// TIA Portal project "Mmot_20230531_1041" (V15.1)

(* hardware
DEVICE "S7-1200 station_1"  S7-1200 Station
   slot 0: "Rack_0"  S7-1200 Rack  Rack  V1.0
   slot 1: "PLC_1"  CPU 1214C DC/DC/DC  6ES7 214-1AG40-0XB0  V4.3
   slot 2: "DI 8x24VDC_1"  6ES7 221-1BF32-0XB0  V2.0
*)

// ===== PLC "PLC_1"  CPU 1214C DC/DC/DC =====

VAR_GLOBAL   // PLC tag table "Default tag table"
   "System_Byte" AT %MB1 : Byte;
   "FirstScan" AT %M1.0 : Bool;
   "DiagStatusUpdate" AT %M1.1 : Bool;
   "AlwaysTRUE" AT %M1.2 : Bool;
   "AlwaysFALSE" AT %M1.3 : Bool;
   "Clock_Byte" AT %MB0 : Byte;
   "Clock_10Hz" AT %M0.0 : Bool;
   "Clock_5Hz" AT %M0.1 : Bool;
   "Clock_2.5Hz" AT %M0.2 : Bool;
   "Clock_2Hz" AT %M0.3 : Bool;
   "Clock_1.25Hz" AT %M0.4 : Bool;
   "Clock_1Hz" AT %M0.5 : Bool;
   "Clock_0.625Hz" AT %M0.6 : Bool;
   "Clock_0.5Hz" AT %M0.7 : Bool;
   "Detector_Axis_Step" AT %Q0.3 : Bool;
   "Doors_Axis_Pulse" AT %Q0.0 : Bool;
   "start" AT %M3.0 : Bool;
   "button_forward" AT %I1.2 : Bool;
   "button_back" AT %I1.3 : Bool;
   "Detector_Axis_Direction" AT %Q0.5 : Bool;
   "Source_Axis_Pulse" AT %Q0.2 : Bool;
   "Source_Axis_Direction" AT %Q0.4 : Bool;
   "Doors_Axis_Direction" AT %Q0.6 : Bool;
   "Roll_Axis_Pulse" AT %Q0.1 : Bool;
   "Roll_Axis_Direction" AT %Q0.7 : Bool;
   "MEMO-1" AT %M10.1 : Bool;
   "MEMO-2" AT %M10.2 : Bool;
END_VAR

VAR_GLOBAL   // PLC tag table "SwitchLimits"
   "SL3A" AT %I0.5 : Bool;
   "SL3B" AT %I0.6 : Bool;
   "SL1A" AT %I0.0 : Bool;
   "SL1B" AT %I0.1 : Bool;
   "SL1C" AT %I0.2 : Bool;
   "SL2A" AT %I0.3 : Bool;
   "SL2B" AT %I0.4 : Bool;
   "SL4A" AT %I0.7 : Bool;
   "SL5" AT %I8.4 : Bool;
   "SL6" AT %I8.5 : Bool;
END_VAR

VAR_GLOBAL   // PLC tag table "source_control"
   "source_block" AT %Q1.0 : Bool;
   "radiation_lamp" AT %Q1.1 : Bool;
   "power_enabled" AT %I1.4 : Bool;
   "emitting" AT %I1.5 : Bool;
END_VAR

VAR_GLOBAL   // PLC tag table "general"
   "S1_alarm" AT %I8.0 : Bool;
   "S2_alarm" AT %I8.1 : Bool;
   "S3_alarm" AT %I8.2 : Bool;
   "S4_alarm" AT %I8.3 : Bool;
   "Q1_control" AT %I1.0 : Bool;
   "Q2_control" AT %I1.1 : Bool;
   "E_button_pressed" AT %M10.0 : Bool;
   "moveC" AT %MW10 : Int;
END_VAR

TYPE "TCON_IP_v42"
   STRUCT
      InterfaceID : Hw_Any;
      ID : Conn_Ouc;
      ConnectionType : Byte := 11;
      ActiveEstablished : Bool := FALSE;
      RemoteAddress : Array[1..4] of Byte;
      RemotePort : UInt := 0;
      LocalPort : UInt := 502;
   END_STRUCT;
   // RemoteAddress[1] := 0;
   // RemoteAddress[2] := 0;
   // RemoteAddress[3] := 0;
   // RemoteAddress[4] := 0;
END_TYPE

DATA_BLOCK "MB_Regs"   // DB2
{ S7_Optimized_Access := 'FALSE' }
VERSION : 0.1
   VAR
      data : Array[0..79] of Word;
   END_VAR
BEGIN
   data[0] := 1;   // 1 Вкл, 0 Выкл
   data[1] := 0;   // 1 - калибровка
   data[2] := 0;   // вращение туда
   data[3] := 0;   // вращение сюда
   data[4] := 0;   // Позиция ст слово
   // data[5] : Позиция мл Слово
   // data[6] : Скорость
   // data[8] : Тек поз ст
   // data[9] : Тек поз мл
   // data[10] : Статус
   // data[11] : Ошибка
   // data[12] : Калибровано
   // data[7] : Сброс
   // data[13] : Halt
   // data[14] : move_to_abs_pos
   // data[15] : move_to_rel_pos
   // data[20] : 1 Вкл, 0 Выкл
   // data[21] : 1 - калибровка
   // data[22] : вращение туда
   // data[23] : вращение сюда
   // data[24] : Позиция ст слово
   // data[25] : Позиция мл Слово
   // data[26] : Скорость
   // data[27] : Сброс
   // data[28] : Тек поз ст
   // data[29] : Тек поз мл
   // data[30] : Статус
   // data[31] : Ошибка
   // data[32] : Калибровано
   // data[33] : Halt
   // data[34] : move_to_abs_pos
   // data[35] : move_to_rel_pos
   // data[40] : 1 Вкл, 0 Выкл
   // data[41] : 1 - калибровка
   // data[42] : вращение туда
   // data[43] : вращение сюда
   // data[44] : Позиция ст слово
   // data[45] : Позиция мл Слово
   // data[46] : Скорость
   // data[47] : Сброс
   // data[48] : Тек поз ст
   // data[49] : Тек поз мл
   // data[50] : Статус
   // data[51] : Ошибка
   // data[52] : Калибровано
   // data[53] : Halt
   // data[54] : move_to_abs_pos
   // data[55] : move_to_rel_pos
   // data[60] : 1 Вкл, 0 Выкл
   // data[61] : 1 - калибровка
   // data[62] : вращение туда
   // data[63] : вращение сюда
   // data[64] : Позиция ст слово
   // data[65] : Позиция мл Слово
   // data[66] : Скорость
   // data[67] : Сброс
   // data[68] : Тек поз ст
   // data[69] : Тек поз мл
   // data[70] : Статус
   // data[71] : Ошибка
   // data[72] : Калибровано
   // data[73] : Halt
   // data[74] : move_to_abs_pos
   // data[75] : move_to_rel_pos
   // data[19] : Block_is_active
   // data[16] : Emission_active
   // data[17] : Power_enabled
   // data[18] : E_stop_button_pressed
   // data[36] : limit1
   // data[37] : limit2
   // data[56] : limit1
   // data[57] : limit2
   // data[76] : moveFrame
   // data[77] : moveCounter
END_DATA_BLOCK

DATA_BLOCK "connect"   // DB3
{ S7_Optimized_Access := 'TRUE' }
VERSION : 0.1
   VAR
      con : "TCON_IP_v42";
      connect : TCON_IP_v4;
   END_VAR
BEGIN
   con.InterfaceID := 64;
   con.ID := 1;
   connect.InterfaceId := 64;
   connect.ID := 1;
   connect.ConnectionType := 11;
   connect.LocalPort := 502;
END_DATA_BLOCK

DATA_BLOCK "door_axe_DB"   // DB6
{ S7_Optimized_Access := 'TRUE' }
VERSION : 0.1
// stored: InstanceOfName door_axe
"door_axe"
BEGIN
END_DATA_BLOCK

DATA_BLOCK "TCP_motion_control_DB"   // DB14
{ S7_Optimized_Access := 'TRUE' }
VERSION : 0.1
// stored: InstanceOfName TCP_motion_control
"TCP_motion_control"
BEGIN
END_DATA_BLOCK

DATA_BLOCK "detector_axe_DB"   // DB15
{ S7_Optimized_Access := 'TRUE' }
VERSION : 0.1
// stored: InstanceOfName detector_axe
"detector_axe"
BEGIN
END_DATA_BLOCK

DATA_BLOCK "source_axe_DB"   // DB17
{ S7_Optimized_Access := 'TRUE' }
VERSION : 0.1
// stored: InstanceOfName source_axe
"source_axe"
BEGIN
END_DATA_BLOCK

DATA_BLOCK "roll_axe_DB"   // DB38
{ S7_Optimized_Access := 'TRUE' }
VERSION : 0.1
// stored: InstanceOfName roll_axe
"roll_axe"
BEGIN
END_DATA_BLOCK

DATA_BLOCK "safety_DB"   // DB40
{ S7_Optimized_Access := 'TRUE' }
VERSION : 0.1
// stored: InstanceOfName safety
"safety"
BEGIN
END_DATA_BLOCK

DATA_BLOCK "CalibrationData"   // DB41
{ S7_Optimized_Access := 'FALSE' }
VERSION : 0.1
   VAR
      Axe1_calibrated : Bool;
      Axe2_calibrated : Bool;
      Axe3_calibrated : Bool;
      Axe4_calibrated : Bool;
      Axe1_saved_pos : Real;
      Axe2_saved_pos : Real;
      Axe3_saved_pos : Real;
      Axe4_saved_pos : Real;
   END_VAR
BEGIN
END_DATA_BLOCK

DATA_BLOCK "safe_done"   // DB47
{ S7_Optimized_Access := 'TRUE' }
VERSION : 0.1
   VAR
      Axe1_SU_calibration_done : Bool;
      Axe2_SU_calibration_done : Bool;
      Axe3_SU_calibration_done : Bool;
      Axe4_SU_calibration_done : Bool;
      control_position : Real;
      control_position_1 : Real;
      control_position_2 : Real;
   END_VAR
BEGIN
END_DATA_BLOCK

// folder: System blocks/Program resources

DATA_BLOCK "IEC_Timer_0_DB"   // DB46
{ S7_Optimized_Access := 'TRUE' }
AUTHOR : Simatic
FAMILY : IEC
NAME : IEC_TMR
VERSION : 1.0
// stored: InstanceOfName IEC_TIMER
"IEC_TIMER"
BEGIN
END_DATA_BLOCK

DATA_BLOCK "IEC_Timer_0_DB_2"   // DB48
{ S7_Optimized_Access := 'TRUE' }
AUTHOR : Simatic
FAMILY : IEC
NAME : IEC_TMR
VERSION : 1.0
// stored: InstanceOfName IEC_TIMER
"IEC_TIMER"
BEGIN
END_DATA_BLOCK

// folder: (top level)

DATA_BLOCK "Detector_Axis"   // DB4, Motion_DB
{ S7_Optimized_Access := 'TRUE' }
AUTHOR : SIMATIC
FAMILY : BasicMC
NAME : TO_PosAx
VERSION : 6.0
// stored: InstanceOfName TO_PositioningAxis
"TO_PositioningAxis"
BEGIN
   // Axis.PassiveHomingReferencePointSwitch_AddressCU = %I0.5
   // Axis.HomingReferencePointSwitch_AddressCU = %I0.5
   // Axis.PositionLimitsMax_AddressCU = %I0.6
   // Axis.PositionLimitsMin_AddressCU = %I0.7
   // Axis.DirectionOutputEnabledCU = TRUE
   // Axis.OnlinePtoIndexCU = 2
   // Axis.LengthUnitNormalized.Distance = 1013
   // Axis.OnlinePtoModeCU = 16#0000_0002
   // Axis.SelectedChannel2EnumCU = %Q0.5
   // Axis.SelectedChannel1EnumCU = %Q0.3
   // Pulse.MinDeltaDeltaFrequencyCU = 0.004
   // Pulse.MaxDeltaDeltaFrequencyCU = 1.0E+10
   // Pulse.MinDeltaFrequencyCU = 0.005
   // Pulse.MaxDeltaFrequencyCU = 9.5E+9
   // Pulse.MinFrequencyCU = 1.0
   // Pulse.MaxFrequencyCU = 100000.0
   // Pulse.OutputSourceCU = 16#0000_0000
   // Axis.SelectPTO = 2
END_DATA_BLOCK

DATA_BLOCK "Source_Axis"   // DB5, Motion_DB
{ S7_Optimized_Access := 'TRUE' }
AUTHOR : SIMATIC
FAMILY : BasicMC
NAME : TO_PosAx
VERSION : 6.0
// stored: InstanceOfName TO_PositioningAxis
"TO_PositioningAxis"
BEGIN
   // Axis.PositionLimitsMax_AddressCU = %I0.4
   // Axis.HomingReferencePointSwitch_AddressCU = %I0.3
   // Axis.PassiveHomingReferencePointSwitch_AddressCU = %I0.3
   // Axis.PositionLimitsMin_AddressCU = %I0.3
   // Axis.DirectionOutputEnabledCU = TRUE
   // Axis.OnlinePtoIndexCU = 1
   // Axis.LengthUnitNormalized.Distance = 1013
   // Axis.OnlinePtoModeCU = 16#0000_0002
   // Axis.SelectedChannel2EnumCU = %Q0.4
   // Axis.SelectedChannel1EnumCU = %Q0.2
   // Pulse.MinDeltaDeltaFrequencyCU = 0.004
   // Pulse.MaxDeltaDeltaFrequencyCU = 1.0E+10
   // Pulse.MinDeltaFrequencyCU = 0.005
   // Pulse.MaxDeltaFrequencyCU = 9.5E+9
   // Pulse.MinFrequencyCU = 1.0
   // Pulse.MaxFrequencyCU = 100000.0
   // Pulse.OutputSourceCU = 16#0000_0000
   // Axis.SelectPTO = 1
END_DATA_BLOCK

DATA_BLOCK "Doors_Axis"   // DB16, Motion_DB
{ S7_Optimized_Access := 'TRUE' }
AUTHOR : SIMATIC
FAMILY : BasicMC
NAME : TO_PosAx
VERSION : 6.0
// stored: InstanceOfName TO_PositioningAxis
"TO_PositioningAxis"
BEGIN
   // Axis.PositionLimitsMin_AddressCU = %I0.1
   // Axis.PassiveHomingReferencePointSwitch_AddressCU = %I0.1
   // Axis.PositionLimitsMax_AddressCU = %I0.0
   // Axis.HomingReferencePointSwitch_AddressCU = %I0.1
   // Axis.DirectionOutputEnabledCU = TRUE
   // Axis.LengthUnitNormalized.Distance = 1013
   // Axis.OnlinePtoModeCU = 16#0000_0002
   // Axis.SelectedChannel2EnumCU = %Q0.6
   // Axis.SelectedChannel1EnumCU = %Q0.0
   // Pulse.MinDeltaDeltaFrequencyCU = 0.004
   // Pulse.MaxDeltaDeltaFrequencyCU = 1.0E+10
   // Pulse.MinDeltaFrequencyCU = 0.005
   // Pulse.MaxDeltaFrequencyCU = 9.5E+9
   // Pulse.MinFrequencyCU = 1.0
   // Pulse.MaxFrequencyCU = 100000.0
   // Pulse.OutputSourceCU = 16#0000_0000
   // Axis.SelectPTO = 0
END_DATA_BLOCK

DATA_BLOCK "Roll_Axis"   // DB39, Motion_DB
{ S7_Optimized_Access := 'TRUE' }
AUTHOR : SIMATIC
FAMILY : BasicMC
NAME : TO_PosAx
VERSION : 6.0
// stored: InstanceOfName TO_PositioningAxis
"TO_PositioningAxis"
BEGIN
   // Axis.LengthUnit.LastDistance = -1
   // Axis.OnlinePtoIndexCU = 3
   // Axis.DirectionOutputEnabledCU = TRUE
   // Axis.OnlinePtoModeCU = 16#0000_0002
   // Axis.SelectedChannel2EnumCU = %Q0.7
   // Axis.SelectedChannel1EnumCU = %Q0.1
   // Pulse.MinDeltaDeltaFrequencyCU = 0.004
   // Pulse.MaxDeltaDeltaFrequencyCU = 1.0E+10
   // Pulse.MinDeltaFrequencyCU = 0.005
   // Pulse.MaxDeltaFrequencyCU = 9.5E+9
   // Pulse.MinFrequencyCU = 1.0
   // Pulse.MaxFrequencyCU = 100000.0
   // Pulse.OutputSourceCU = 16#0000_0000
   // Axis.SelectPTO = 3
END_DATA_BLOCK

FUNCTION_BLOCK "TCP_motion_control"   // FB1, LAD
{ S7_Optimized_Access := 'TRUE' }
VERSION : 0.1
   VAR_TEMP
      temp_vel : UDInt;
      temp_vel_real : Real;
      temp_val2 : Real;
   END_VAR
   VAR_TEMP   // added for the SCL form of the ladder/FBD networks
      _w1 : Bool;
   END_VAR
BEGIN

REGION Network 1
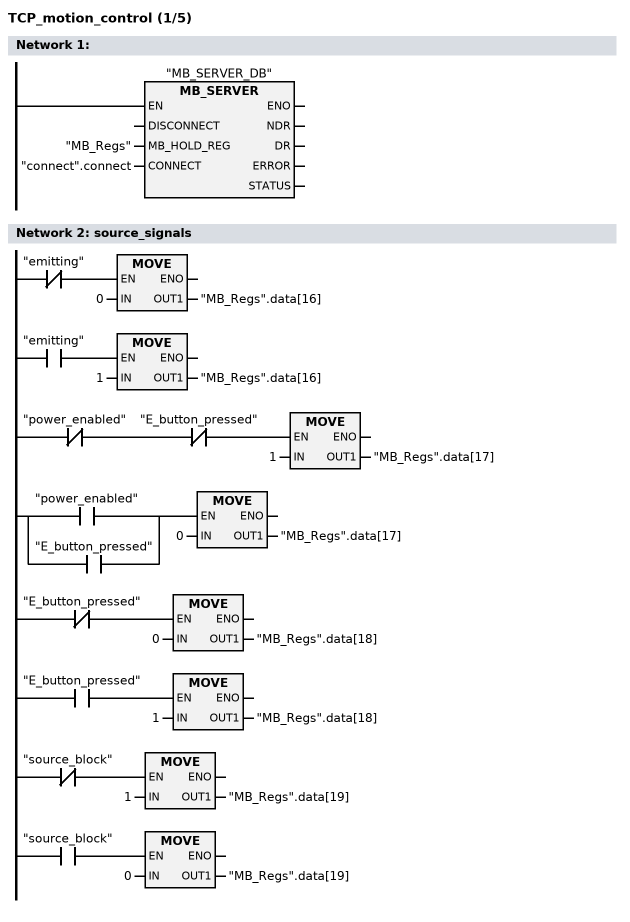
   "MB_SERVER_DB"(MB_HOLD_REG := "MB_Regs", CONNECT := "connect".connect);   // MB_SERVER
END_REGION

REGION Network 2: source_signals
   RUNG wire#powerrail
      I_Contact( "emitting" )
      Move(in := 0, out1 => "MB_Regs".data[16])
   END_RUNG
   RUNG wire#powerrail
      Contact( "emitting" )
      Move(in := 1, out1 => "MB_Regs".data[16])
   END_RUNG
   RUNG wire#powerrail
      I_Contact( "power_enabled" )
      I_Contact( "E_button_pressed" )
      Move(in := 1, out1 => "MB_Regs".data[17])
   END_RUNG
   RUNG wire#powerrail
      Contact( "power_enabled" )
      wire#w1
      Move(in := 0, out1 => "MB_Regs".data[17])
   END_RUNG
   RUNG wire#powerrail
      Contact( "E_button_pressed" )
   END_RUNG wire#w1
   RUNG wire#powerrail
      I_Contact( "E_button_pressed" )
      Move(in := 0, out1 => "MB_Regs".data[18])
   END_RUNG
   RUNG wire#powerrail
      Contact( "E_button_pressed" )
      Move(in := 1, out1 => "MB_Regs".data[18])
   END_RUNG
   RUNG wire#powerrail
      I_Contact( "source_block" )
      Move(in := 1, out1 => "MB_Regs".data[19])
   END_RUNG
   RUNG wire#powerrail
      Contact( "source_block" )
      Move(in := 0, out1 => "MB_Regs".data[19])
   END_RUNG
   // the same network as SCL:
   IF NOT "emitting" THEN "MB_Regs".data[16] := 0; END_IF;
   IF "emitting" THEN "MB_Regs".data[16] := 1; END_IF;
   IF NOT "power_enabled" AND NOT "E_button_pressed" THEN "MB_Regs".data[17] := 1; END_IF;
   IF "power_enabled" OR "E_button_pressed" THEN "MB_Regs".data[17] := 0; END_IF;
   IF NOT "E_button_pressed" THEN "MB_Regs".data[18] := 0; END_IF;
   IF "E_button_pressed" THEN "MB_Regs".data[18] := 1; END_IF;
   IF NOT "source_block" THEN "MB_Regs".data[19] := 1; END_IF;
   IF "source_block" THEN "MB_Regs".data[19] := 0; END_IF;
END_REGION

REGION Network 3: Motor 1 doors
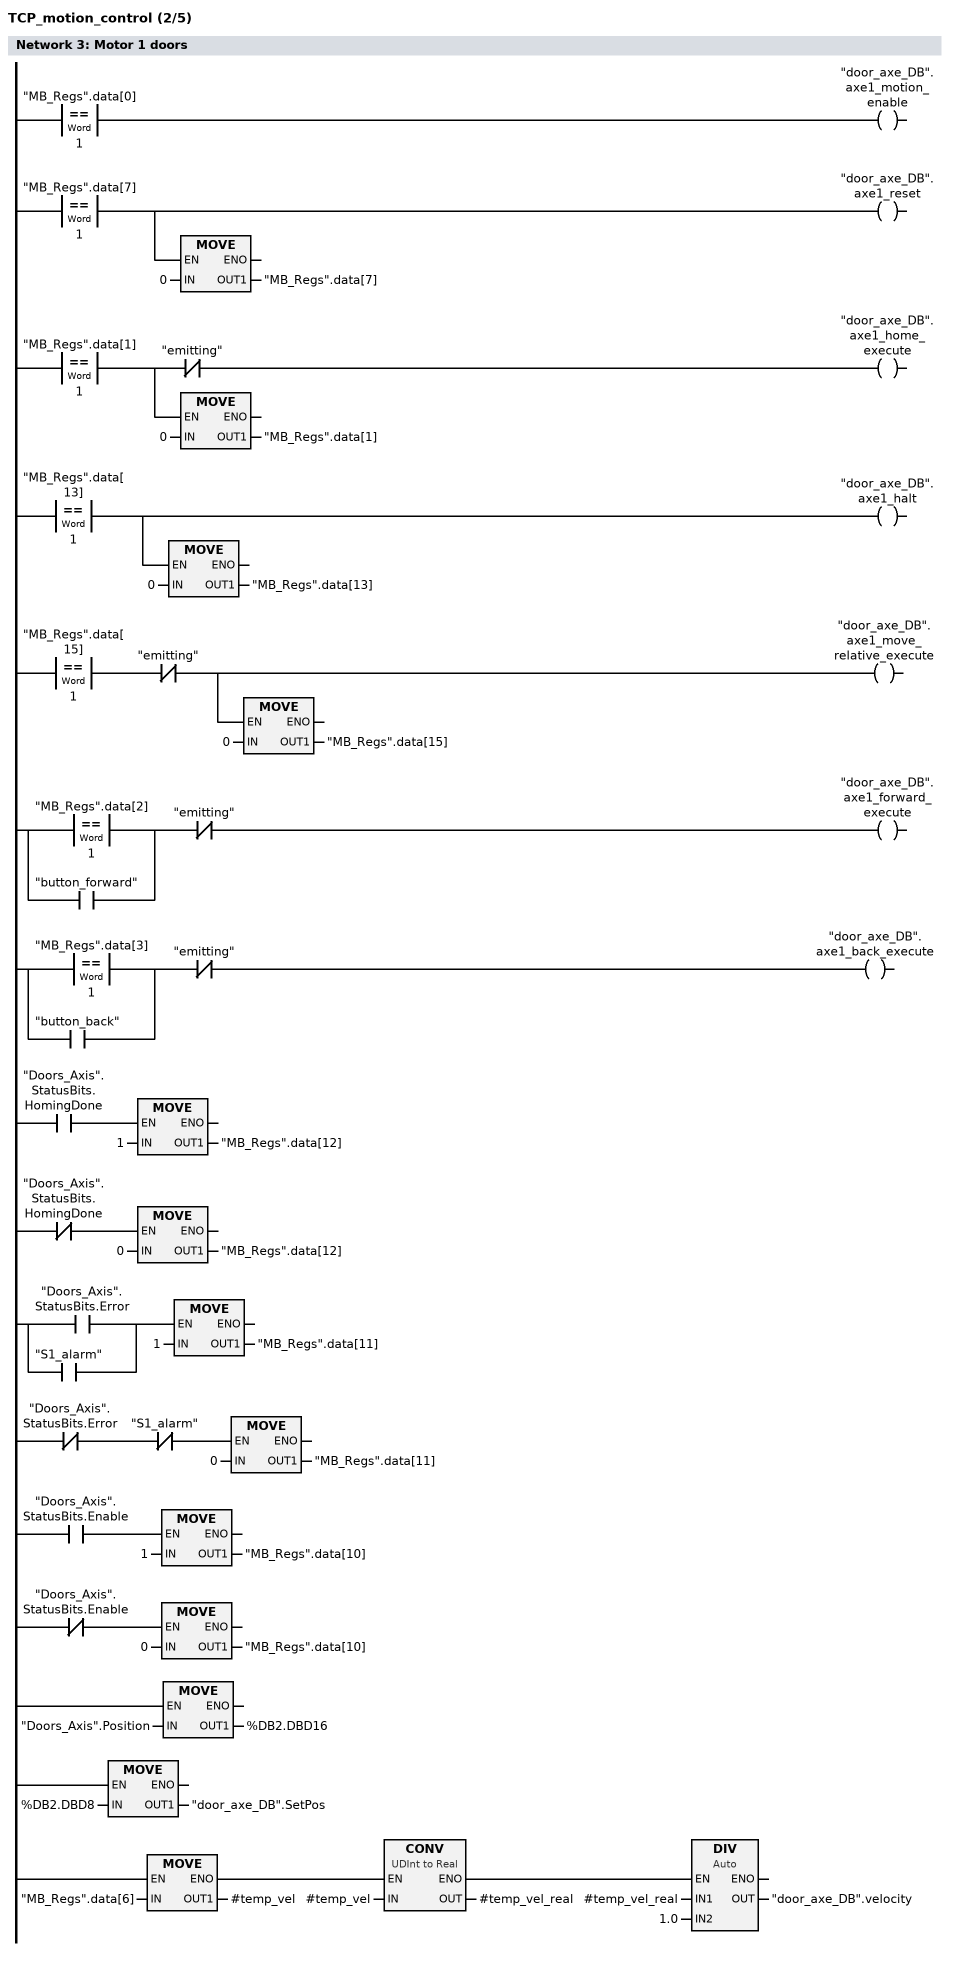
   RUNG wire#powerrail
      { S7_Templates := "SrcType := Word" } EQ_Contact(in1 := "MB_Regs".data[0], in2 := 1)
      Coil( "door_axe_DB".axe1_motion_enable )
   END_RUNG
   RUNG wire#powerrail
      { S7_Templates := "SrcType := Word" } EQ_Contact(in1 := "MB_Regs".data[7], in2 := 1)
      wire#w1
      Coil( "door_axe_DB".axe1_reset )
   END_RUNG
   RUNG wire#w1
      Move(in := 0, out1 => "MB_Regs".data[7])
   END_RUNG
   RUNG wire#powerrail
      { S7_Templates := "SrcType := Word" } EQ_Contact(in1 := "MB_Regs".data[1], in2 := 1)
      wire#w2
      I_Contact( "emitting" )
      Coil( "door_axe_DB".axe1_home_execute )
   END_RUNG
   RUNG wire#w2
      Move(in := 0, out1 => "MB_Regs".data[1])
   END_RUNG
   RUNG wire#powerrail
      { S7_Templates := "SrcType := Word" } EQ_Contact(in1 := "MB_Regs".data[13], in2 := 1)
      wire#w3
      Coil( "door_axe_DB".axe1_halt )
   END_RUNG
   RUNG wire#w3
      Move(in := 0, out1 => "MB_Regs".data[13])
   END_RUNG
   RUNG wire#powerrail
      { S7_Templates := "SrcType := Word" } EQ_Contact(in1 := "MB_Regs".data[15], in2 := 1)
      I_Contact( "emitting" )
      wire#w4
      Coil( "door_axe_DB".axe1_move_relative_execute )
   END_RUNG
   RUNG wire#w4
      Move(in := 0, out1 => "MB_Regs".data[15])
   END_RUNG
   RUNG wire#powerrail
      { S7_Templates := "SrcType := Word" } EQ_Contact(in1 := "MB_Regs".data[2], in2 := 1)
      wire#w5
      I_Contact( "emitting" )
      Coil( "door_axe_DB".axe1_forward_execute )
   END_RUNG
   RUNG wire#powerrail
      Contact( "button_forward" )
   END_RUNG wire#w5
   RUNG wire#powerrail
      { S7_Templates := "SrcType := Word" } EQ_Contact(in1 := "MB_Regs".data[3], in2 := 1)
      wire#w6
      I_Contact( "emitting" )
      Coil( "door_axe_DB".axe1_back_execute )
   END_RUNG
   RUNG wire#powerrail
      Contact( "button_back" )
   END_RUNG wire#w6
   RUNG wire#powerrail
      Contact( "Doors_Axis".StatusBits.HomingDone )
      Move(in := 1, out1 => "MB_Regs".data[12])
   END_RUNG
   RUNG wire#powerrail
      I_Contact( "Doors_Axis".StatusBits.HomingDone )
      Move(in := 0, out1 => "MB_Regs".data[12])
   END_RUNG
   RUNG wire#powerrail
      Contact( "Doors_Axis".StatusBits.Error )
      wire#w7
      Move(in := 1, out1 => "MB_Regs".data[11])
   END_RUNG
   RUNG wire#powerrail
      Contact( "S1_alarm" )
   END_RUNG wire#w7
   RUNG wire#powerrail
      I_Contact( "Doors_Axis".StatusBits.Error )
      I_Contact( "S1_alarm" )
      Move(in := 0, out1 => "MB_Regs".data[11])
   END_RUNG
   RUNG wire#powerrail
      Contact( "Doors_Axis".StatusBits.Enable )
      Move(in := 1, out1 => "MB_Regs".data[10])
   END_RUNG
   RUNG wire#powerrail
      I_Contact( "Doors_Axis".StatusBits.Enable )
      Move(in := 0, out1 => "MB_Regs".data[10])
   END_RUNG
   RUNG wire#powerrail
      Move(in := "Doors_Axis".Position, out1 => %DB2.DBD16)
   END_RUNG
   RUNG wire#powerrail
      Move(in := %DB2.DBD8, out1 => "door_axe_DB".SetPos)
   END_RUNG
   RUNG wire#powerrail
      Move(in := "MB_Regs".data[6], out1 => #temp_vel)
      { S7_Templates := "[SrcType := UDInt, DestType := Real]" } Convert(in := #temp_vel, out => #temp_vel_real)
      Div(in1 := #temp_vel_real, in2 := 1.0, out => "door_axe_DB".velocity)
   END_RUNG
   // the same network as SCL:
   "door_axe_DB".axe1_motion_enable := "MB_Regs".data[0] = 1;
   "door_axe_DB".axe1_reset := "MB_Regs".data[7] = 1;
   IF "door_axe_DB".axe1_reset THEN "MB_Regs".data[7] := 0; END_IF;
   #_w1 := "MB_Regs".data[1] = 1;
   "door_axe_DB".axe1_home_execute := #_w1 AND NOT "emitting";
   IF #_w1 THEN "MB_Regs".data[1] := 0; END_IF;
   "door_axe_DB".axe1_halt := "MB_Regs".data[13] = 1;
   IF "door_axe_DB".axe1_halt THEN "MB_Regs".data[13] := 0; END_IF;
   "door_axe_DB".axe1_move_relative_execute := ("MB_Regs".data[15] = 1) AND NOT "emitting";
   IF "door_axe_DB".axe1_move_relative_execute THEN "MB_Regs".data[15] := 0; END_IF;
   "door_axe_DB".axe1_forward_execute := (("MB_Regs".data[2] = 1) OR "button_forward") AND NOT "emitting";
   "door_axe_DB".axe1_back_execute := (("MB_Regs".data[3] = 1) OR "button_back") AND NOT "emitting";
   IF "Doors_Axis".StatusBits.HomingDone THEN "MB_Regs".data[12] := 1; END_IF;
   IF NOT "Doors_Axis".StatusBits.HomingDone THEN "MB_Regs".data[12] := 0; END_IF;
   IF "Doors_Axis".StatusBits.Error OR "S1_alarm" THEN "MB_Regs".data[11] := 1; END_IF;
   IF NOT "Doors_Axis".StatusBits.Error AND NOT "S1_alarm" THEN "MB_Regs".data[11] := 0; END_IF;
   IF "Doors_Axis".StatusBits.Enable THEN "MB_Regs".data[10] := 1; END_IF;
   IF NOT "Doors_Axis".StatusBits.Enable THEN "MB_Regs".data[10] := 0; END_IF;
   %DB2.DBD16 := "Doors_Axis".Position;
   "door_axe_DB".SetPos := %DB2.DBD8;
   #temp_vel := "MB_Regs".data[6];
   #temp_vel_real := UDINT_TO_REAL(#temp_vel);
   "door_axe_DB".velocity := #temp_vel_real / 1.0;
END_REGION

REGION Network 4: Motor 2 source
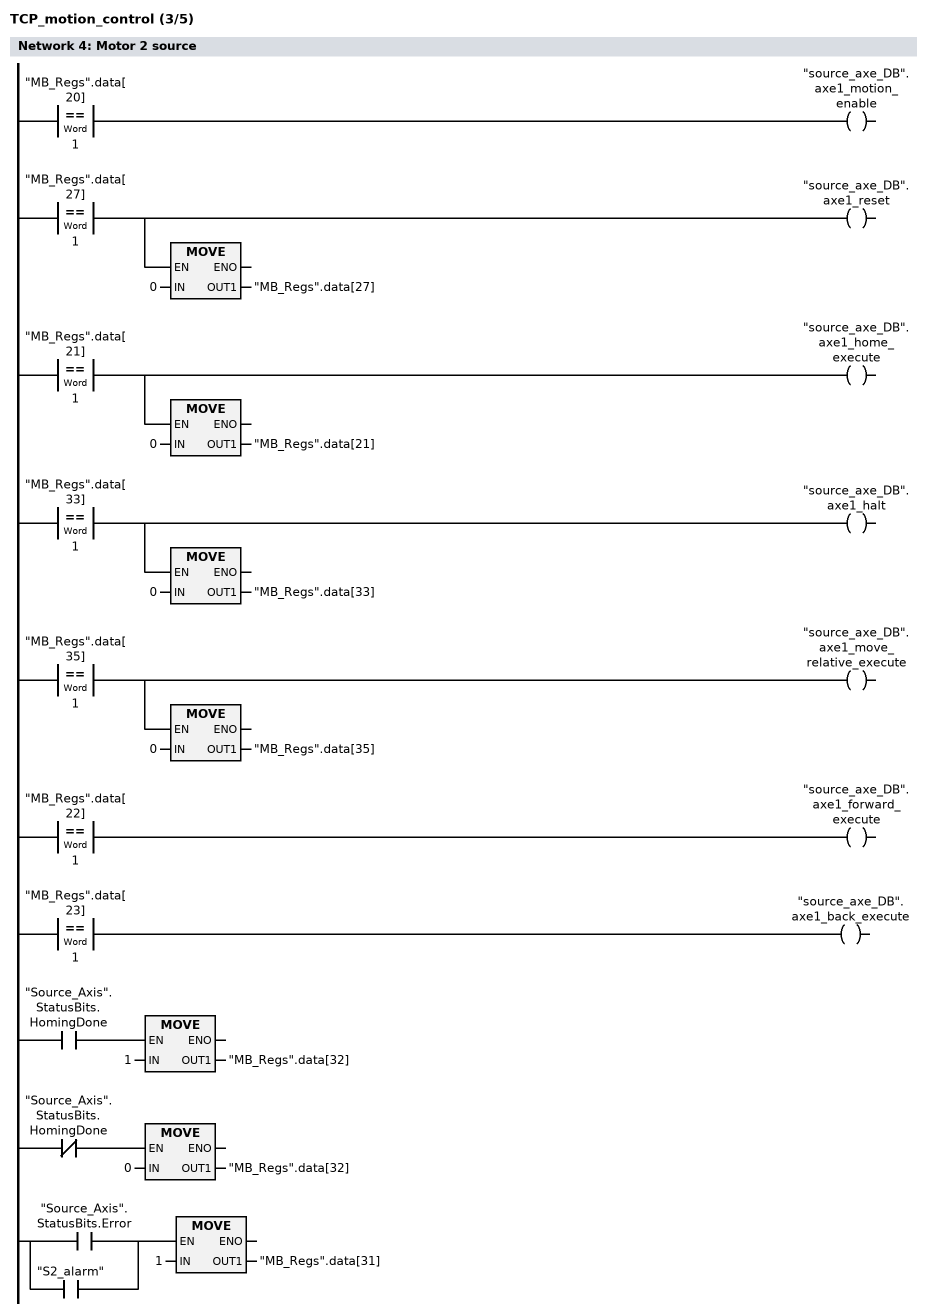
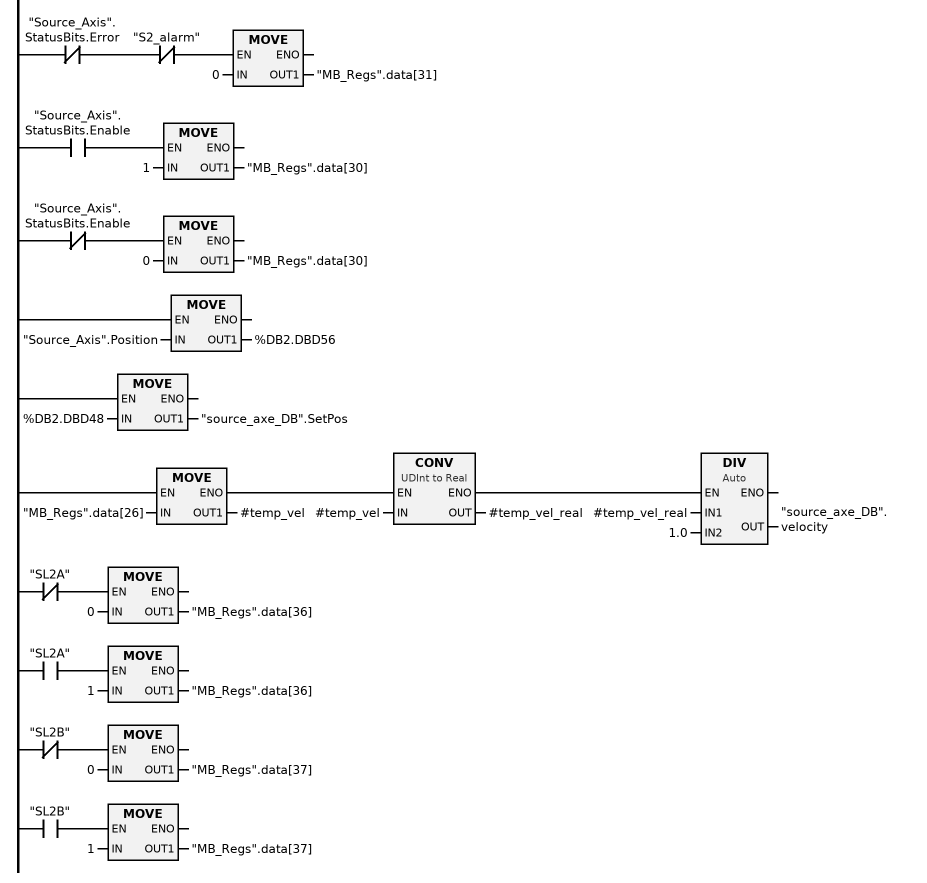
   RUNG wire#powerrail
      { S7_Templates := "SrcType := Word" } EQ_Contact(in1 := "MB_Regs".data[20], in2 := 1)
      Coil( "source_axe_DB".axe1_motion_enable )
   END_RUNG
   RUNG wire#powerrail
      { S7_Templates := "SrcType := Word" } EQ_Contact(in1 := "MB_Regs".data[27], in2 := 1)
      wire#w1
      Coil( "source_axe_DB".axe1_reset )
   END_RUNG
   RUNG wire#w1
      Move(in := 0, out1 => "MB_Regs".data[27])
   END_RUNG
   RUNG wire#powerrail
      { S7_Templates := "SrcType := Word" } EQ_Contact(in1 := "MB_Regs".data[21], in2 := 1)
      wire#w2
      Coil( "source_axe_DB".axe1_home_execute )
   END_RUNG
   RUNG wire#w2
      Move(in := 0, out1 => "MB_Regs".data[21])
   END_RUNG
   RUNG wire#powerrail
      { S7_Templates := "SrcType := Word" } EQ_Contact(in1 := "MB_Regs".data[33], in2 := 1)
      wire#w3
      Coil( "source_axe_DB".axe1_halt )
   END_RUNG
   RUNG wire#w3
      Move(in := 0, out1 => "MB_Regs".data[33])
   END_RUNG
   RUNG wire#powerrail
      { S7_Templates := "SrcType := Word" } EQ_Contact(in1 := "MB_Regs".data[35], in2 := 1)
      wire#w4
      Coil( "source_axe_DB".axe1_move_relative_execute )
   END_RUNG
   RUNG wire#w4
      Move(in := 0, out1 => "MB_Regs".data[35])
   END_RUNG
   RUNG wire#powerrail
      { S7_Templates := "SrcType := Word" } EQ_Contact(in1 := "MB_Regs".data[22], in2 := 1)
      Coil( "source_axe_DB".axe1_forward_execute )
   END_RUNG
   RUNG wire#powerrail
      { S7_Templates := "SrcType := Word" } EQ_Contact(in1 := "MB_Regs".data[23], in2 := 1)
      Coil( "source_axe_DB".axe1_back_execute )
   END_RUNG
   RUNG wire#powerrail
      Contact( "Source_Axis".StatusBits.HomingDone )
      Move(in := 1, out1 => "MB_Regs".data[32])
   END_RUNG
   RUNG wire#powerrail
      I_Contact( "Source_Axis".StatusBits.HomingDone )
      Move(in := 0, out1 => "MB_Regs".data[32])
   END_RUNG
   RUNG wire#powerrail
      Contact( "Source_Axis".StatusBits.Error )
      wire#w5
      Move(in := 1, out1 => "MB_Regs".data[31])
   END_RUNG
   RUNG wire#powerrail
      Contact( "S2_alarm" )
   END_RUNG wire#w5
   RUNG wire#powerrail
      I_Contact( "Source_Axis".StatusBits.Error )
      I_Contact( "S2_alarm" )
      Move(in := 0, out1 => "MB_Regs".data[31])
   END_RUNG
   RUNG wire#powerrail
      Contact( "Source_Axis".StatusBits.Enable )
      Move(in := 1, out1 => "MB_Regs".data[30])
   END_RUNG
   RUNG wire#powerrail
      I_Contact( "Source_Axis".StatusBits.Enable )
      Move(in := 0, out1 => "MB_Regs".data[30])
   END_RUNG
   RUNG wire#powerrail
      Move(in := "Source_Axis".Position, out1 => %DB2.DBD56)
   END_RUNG
   RUNG wire#powerrail
      Move(in := %DB2.DBD48, out1 => "source_axe_DB".SetPos)
   END_RUNG
   RUNG wire#powerrail
      Move(in := "MB_Regs".data[26], out1 => #temp_vel)
      { S7_Templates := "[SrcType := UDInt, DestType := Real]" } Convert(in := #temp_vel, out => #temp_vel_real)
      Div(in1 := #temp_vel_real, in2 := 1.0, out => "source_axe_DB".velocity)
   END_RUNG
   RUNG wire#powerrail
      I_Contact( "SL2A" )
      Move(in := 0, out1 => "MB_Regs".data[36])
   END_RUNG
   RUNG wire#powerrail
      Contact( "SL2A" )
      Move(in := 1, out1 => "MB_Regs".data[36])
   END_RUNG
   RUNG wire#powerrail
      I_Contact( "SL2B" )
      Move(in := 0, out1 => "MB_Regs".data[37])
   END_RUNG
   RUNG wire#powerrail
      Contact( "SL2B" )
      Move(in := 1, out1 => "MB_Regs".data[37])
   END_RUNG
   // the same network as SCL:
   "source_axe_DB".axe1_motion_enable := "MB_Regs".data[20] = 1;
   "source_axe_DB".axe1_reset := "MB_Regs".data[27] = 1;
   IF "source_axe_DB".axe1_reset THEN "MB_Regs".data[27] := 0; END_IF;
   "source_axe_DB".axe1_home_execute := "MB_Regs".data[21] = 1;
   IF "source_axe_DB".axe1_home_execute THEN "MB_Regs".data[21] := 0; END_IF;
   "source_axe_DB".axe1_halt := "MB_Regs".data[33] = 1;
   IF "source_axe_DB".axe1_halt THEN "MB_Regs".data[33] := 0; END_IF;
   "source_axe_DB".axe1_move_relative_execute := "MB_Regs".data[35] = 1;
   IF "source_axe_DB".axe1_move_relative_execute THEN "MB_Regs".data[35] := 0; END_IF;
   "source_axe_DB".axe1_forward_execute := "MB_Regs".data[22] = 1;
   "source_axe_DB".axe1_back_execute := "MB_Regs".data[23] = 1;
   IF "Source_Axis".StatusBits.HomingDone THEN "MB_Regs".data[32] := 1; END_IF;
   IF NOT "Source_Axis".StatusBits.HomingDone THEN "MB_Regs".data[32] := 0; END_IF;
   IF "Source_Axis".StatusBits.Error OR "S2_alarm" THEN "MB_Regs".data[31] := 1; END_IF;
   IF NOT "Source_Axis".StatusBits.Error AND NOT "S2_alarm" THEN "MB_Regs".data[31] := 0; END_IF;
   IF "Source_Axis".StatusBits.Enable THEN "MB_Regs".data[30] := 1; END_IF;
   IF NOT "Source_Axis".StatusBits.Enable THEN "MB_Regs".data[30] := 0; END_IF;
   %DB2.DBD56 := "Source_Axis".Position;
   "source_axe_DB".SetPos := %DB2.DBD48;
   #temp_vel := "MB_Regs".data[26];
   #temp_vel_real := UDINT_TO_REAL(#temp_vel);
   "source_axe_DB".velocity := #temp_vel_real / 1.0;
   IF NOT "SL2A" THEN "MB_Regs".data[36] := 0; END_IF;
   IF "SL2A" THEN "MB_Regs".data[36] := 1; END_IF;
   IF NOT "SL2B" THEN "MB_Regs".data[37] := 0; END_IF;
   IF "SL2B" THEN "MB_Regs".data[37] := 1; END_IF;
END_REGION

REGION Network 5: Motor 3 (detector)
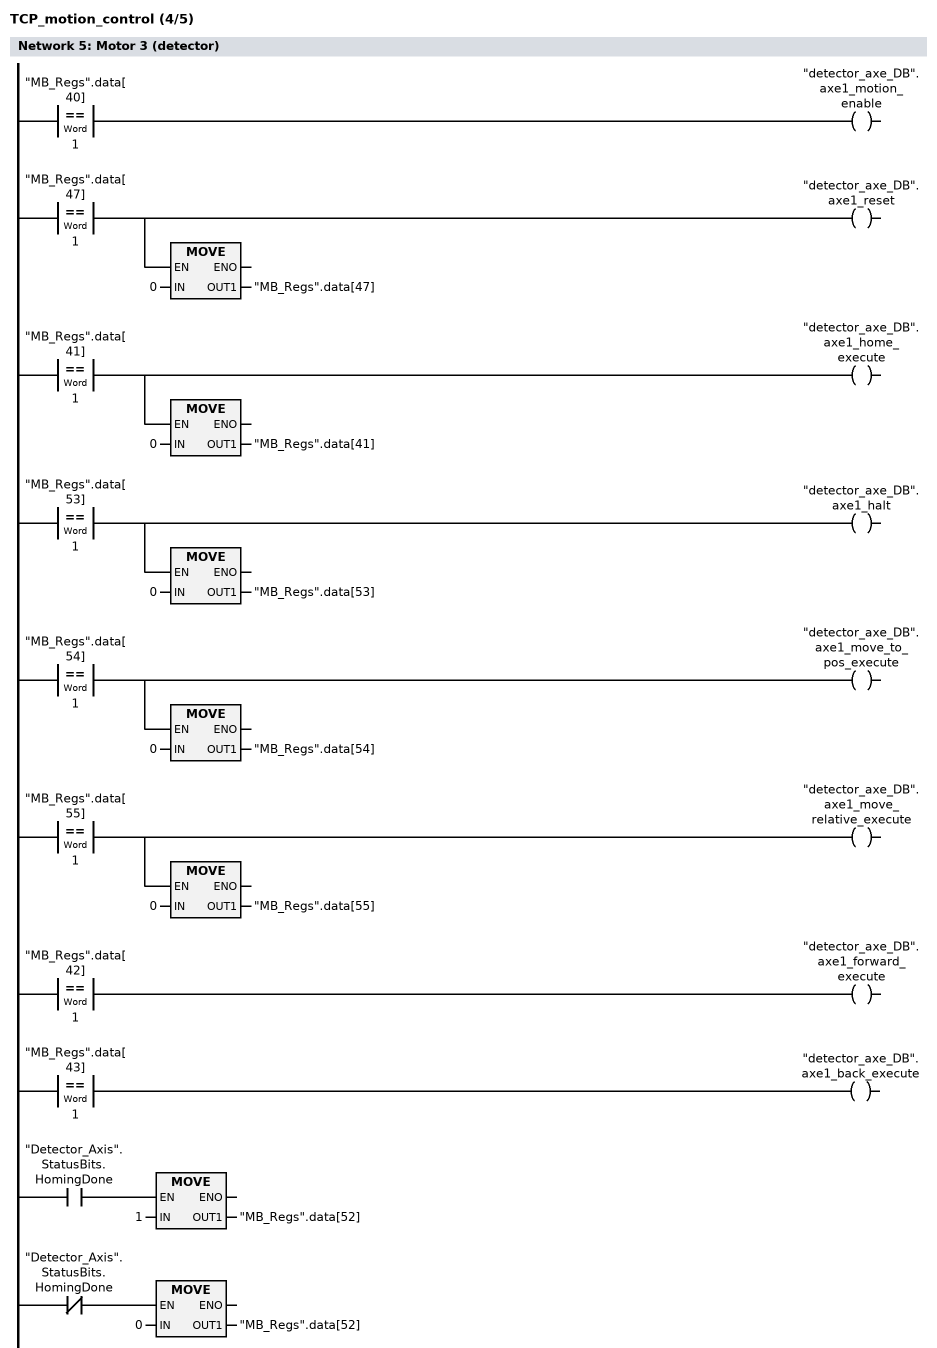
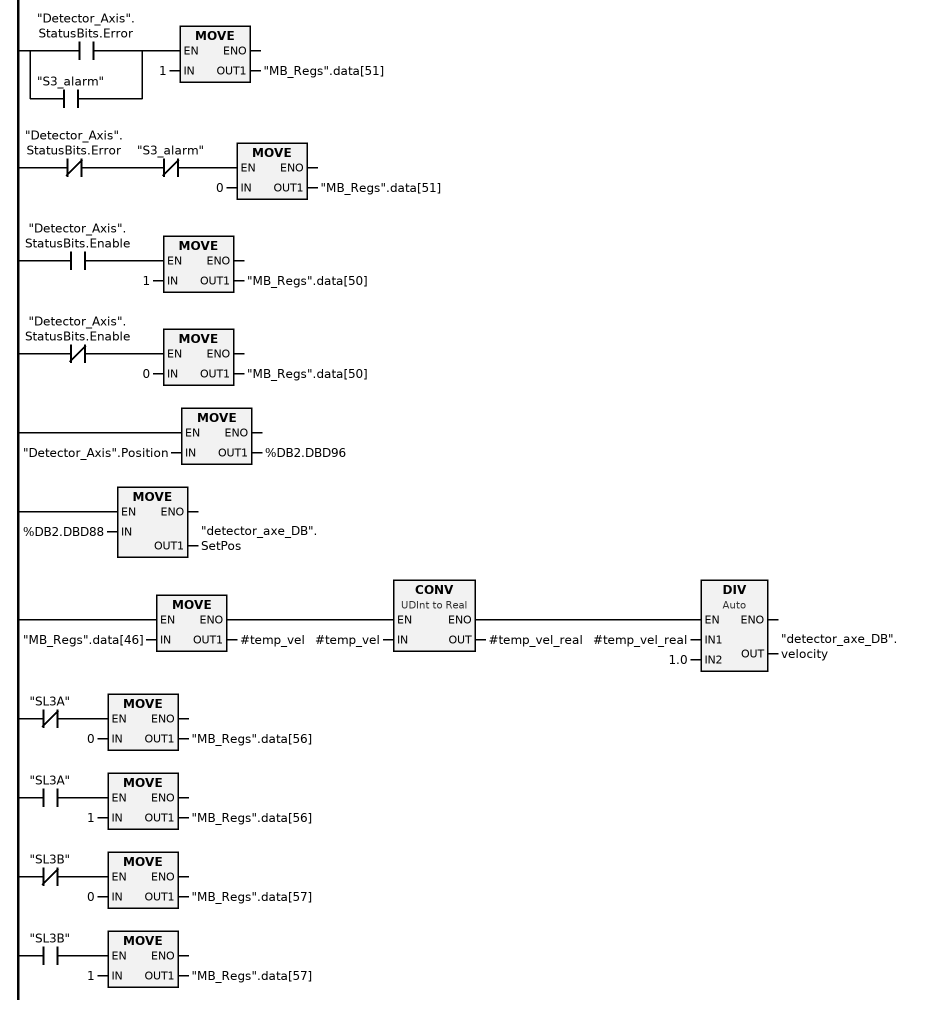
   RUNG wire#powerrail
      { S7_Templates := "SrcType := Word" } EQ_Contact(in1 := "MB_Regs".data[40], in2 := 1)
      Coil( "detector_axe_DB".axe1_motion_enable )
   END_RUNG
   RUNG wire#powerrail
      { S7_Templates := "SrcType := Word" } EQ_Contact(in1 := "MB_Regs".data[47], in2 := 1)
      wire#w1
      Coil( "detector_axe_DB".axe1_reset )
   END_RUNG
   RUNG wire#w1
      Move(in := 0, out1 => "MB_Regs".data[47])
   END_RUNG
   RUNG wire#powerrail
      { S7_Templates := "SrcType := Word" } EQ_Contact(in1 := "MB_Regs".data[41], in2 := 1)
      wire#w2
      Coil( "detector_axe_DB".axe1_home_execute )
   END_RUNG
   RUNG wire#w2
      Move(in := 0, out1 => "MB_Regs".data[41])
   END_RUNG
   RUNG wire#powerrail
      { S7_Templates := "SrcType := Word" } EQ_Contact(in1 := "MB_Regs".data[53], in2 := 1)
      wire#w3
      Coil( "detector_axe_DB".axe1_halt )
   END_RUNG
   RUNG wire#w3
      Move(in := 0, out1 => "MB_Regs".data[53])
   END_RUNG
   RUNG wire#powerrail
      { S7_Templates := "SrcType := Word" } EQ_Contact(in1 := "MB_Regs".data[54], in2 := 1)
      wire#w4
      Coil( "detector_axe_DB".axe1_move_to_pos_execute )
   END_RUNG
   RUNG wire#w4
      Move(in := 0, out1 => "MB_Regs".data[54])
   END_RUNG
   RUNG wire#powerrail
      { S7_Templates := "SrcType := Word" } EQ_Contact(in1 := "MB_Regs".data[55], in2 := 1)
      wire#w5
      Coil( "detector_axe_DB".axe1_move_relative_execute )
   END_RUNG
   RUNG wire#w5
      Move(in := 0, out1 => "MB_Regs".data[55])
   END_RUNG
   RUNG wire#powerrail
      { S7_Templates := "SrcType := Word" } EQ_Contact(in1 := "MB_Regs".data[42], in2 := 1)
      Coil( "detector_axe_DB".axe1_forward_execute )
   END_RUNG
   RUNG wire#powerrail
      { S7_Templates := "SrcType := Word" } EQ_Contact(in1 := "MB_Regs".data[43], in2 := 1)
      Coil( "detector_axe_DB".axe1_back_execute )
   END_RUNG
   RUNG wire#powerrail
      Contact( "Detector_Axis".StatusBits.HomingDone )
      Move(in := 1, out1 => "MB_Regs".data[52])
   END_RUNG
   RUNG wire#powerrail
      I_Contact( "Detector_Axis".StatusBits.HomingDone )
      Move(in := 0, out1 => "MB_Regs".data[52])
   END_RUNG
   RUNG wire#powerrail
      Contact( "Detector_Axis".StatusBits.Error )
      wire#w6
      Move(in := 1, out1 => "MB_Regs".data[51])
   END_RUNG
   RUNG wire#powerrail
      Contact( "S3_alarm" )
   END_RUNG wire#w6
   RUNG wire#powerrail
      I_Contact( "Detector_Axis".StatusBits.Error )
      I_Contact( "S3_alarm" )
      Move(in := 0, out1 => "MB_Regs".data[51])
   END_RUNG
   RUNG wire#powerrail
      Contact( "Detector_Axis".StatusBits.Enable )
      Move(in := 1, out1 => "MB_Regs".data[50])
   END_RUNG
   RUNG wire#powerrail
      I_Contact( "Detector_Axis".StatusBits.Enable )
      Move(in := 0, out1 => "MB_Regs".data[50])
   END_RUNG
   RUNG wire#powerrail
      Move(in := "Detector_Axis".Position, out1 => %DB2.DBD96)
   END_RUNG
   RUNG wire#powerrail
      Move(in := %DB2.DBD88, out1 => "detector_axe_DB".SetPos)
   END_RUNG
   RUNG wire#powerrail
      Move(in := "MB_Regs".data[46], out1 => #temp_vel)
      { S7_Templates := "[SrcType := UDInt, DestType := Real]" } Convert(in := #temp_vel, out => #temp_vel_real)
      Div(in1 := #temp_vel_real, in2 := 1.0, out => "detector_axe_DB".velocity)
   END_RUNG
   RUNG wire#powerrail
      I_Contact( "SL3A" )
      Move(in := 0, out1 => "MB_Regs".data[56])
   END_RUNG
   RUNG wire#powerrail
      Contact( "SL3A" )
      Move(in := 1, out1 => "MB_Regs".data[56])
   END_RUNG
   RUNG wire#powerrail
      I_Contact( "SL3B" )
      Move(in := 0, out1 => "MB_Regs".data[57])
   END_RUNG
   RUNG wire#powerrail
      Contact( "SL3B" )
      Move(in := 1, out1 => "MB_Regs".data[57])
   END_RUNG
   // the same network as SCL:
   "detector_axe_DB".axe1_motion_enable := "MB_Regs".data[40] = 1;
   "detector_axe_DB".axe1_reset := "MB_Regs".data[47] = 1;
   IF "detector_axe_DB".axe1_reset THEN "MB_Regs".data[47] := 0; END_IF;
   "detector_axe_DB".axe1_home_execute := "MB_Regs".data[41] = 1;
   IF "detector_axe_DB".axe1_home_execute THEN "MB_Regs".data[41] := 0; END_IF;
   "detector_axe_DB".axe1_halt := "MB_Regs".data[53] = 1;
   IF "detector_axe_DB".axe1_halt THEN "MB_Regs".data[53] := 0; END_IF;
   "detector_axe_DB".axe1_move_to_pos_execute := "MB_Regs".data[54] = 1;
   IF "detector_axe_DB".axe1_move_to_pos_execute THEN "MB_Regs".data[54] := 0; END_IF;
   "detector_axe_DB".axe1_move_relative_execute := "MB_Regs".data[55] = 1;
   IF "detector_axe_DB".axe1_move_relative_execute THEN "MB_Regs".data[55] := 0; END_IF;
   "detector_axe_DB".axe1_forward_execute := "MB_Regs".data[42] = 1;
   "detector_axe_DB".axe1_back_execute := "MB_Regs".data[43] = 1;
   IF "Detector_Axis".StatusBits.HomingDone THEN "MB_Regs".data[52] := 1; END_IF;
   IF NOT "Detector_Axis".StatusBits.HomingDone THEN "MB_Regs".data[52] := 0; END_IF;
   IF "Detector_Axis".StatusBits.Error OR "S3_alarm" THEN "MB_Regs".data[51] := 1; END_IF;
   IF NOT "Detector_Axis".StatusBits.Error AND NOT "S3_alarm" THEN "MB_Regs".data[51] := 0; END_IF;
   IF "Detector_Axis".StatusBits.Enable THEN "MB_Regs".data[50] := 1; END_IF;
   IF NOT "Detector_Axis".StatusBits.Enable THEN "MB_Regs".data[50] := 0; END_IF;
   %DB2.DBD96 := "Detector_Axis".Position;
   "detector_axe_DB".SetPos := %DB2.DBD88;
   #temp_vel := "MB_Regs".data[46];
   #temp_vel_real := UDINT_TO_REAL(#temp_vel);
   "detector_axe_DB".velocity := #temp_vel_real / 1.0;
   IF NOT "SL3A" THEN "MB_Regs".data[56] := 0; END_IF;
   IF "SL3A" THEN "MB_Regs".data[56] := 1; END_IF;
   IF NOT "SL3B" THEN "MB_Regs".data[57] := 0; END_IF;
   IF "SL3B" THEN "MB_Regs".data[57] := 1; END_IF;
END_REGION

REGION Network 6: Motor 4 (ROLL)
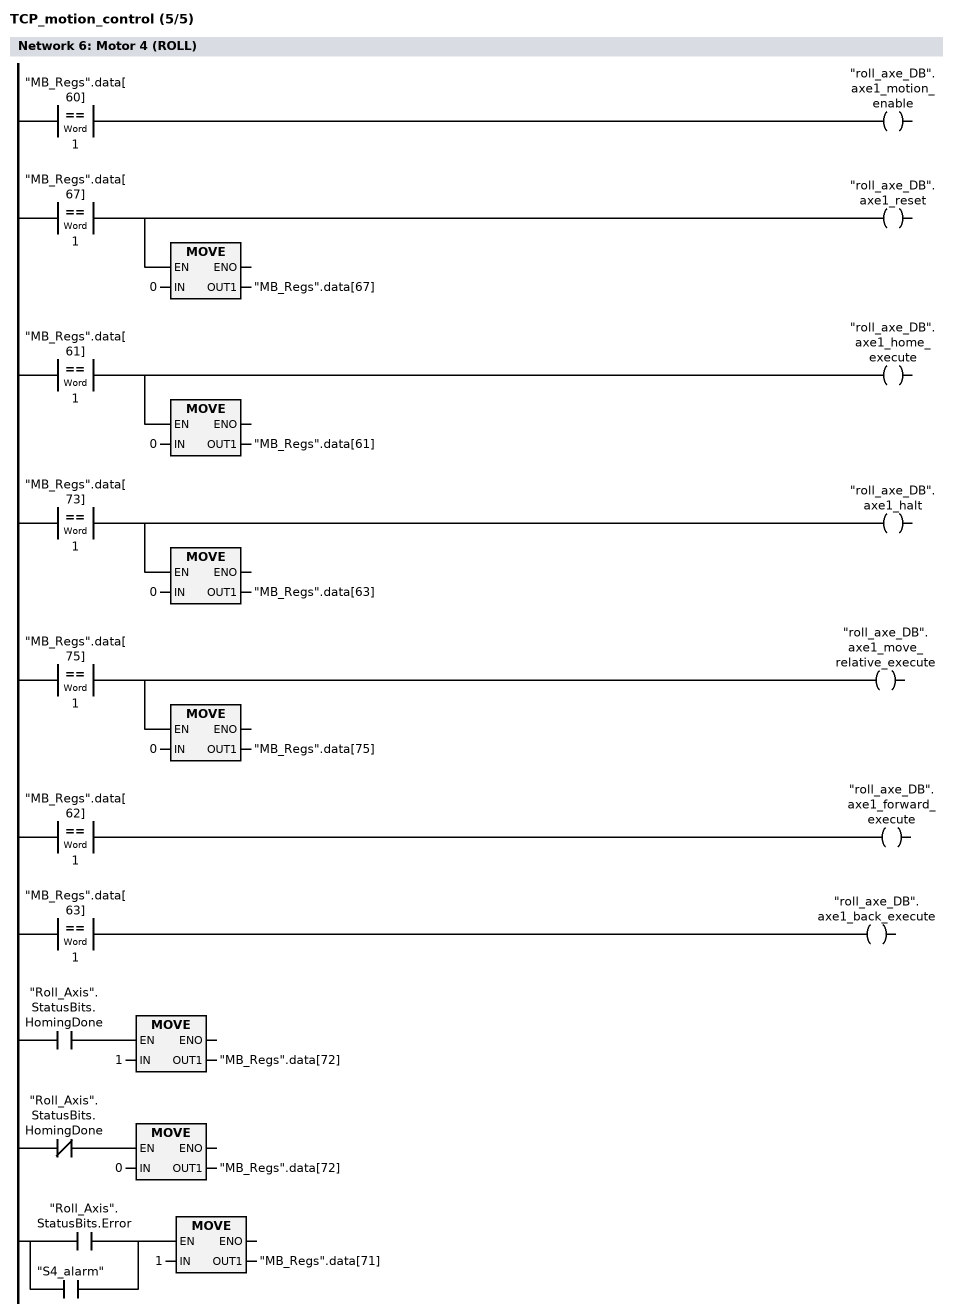
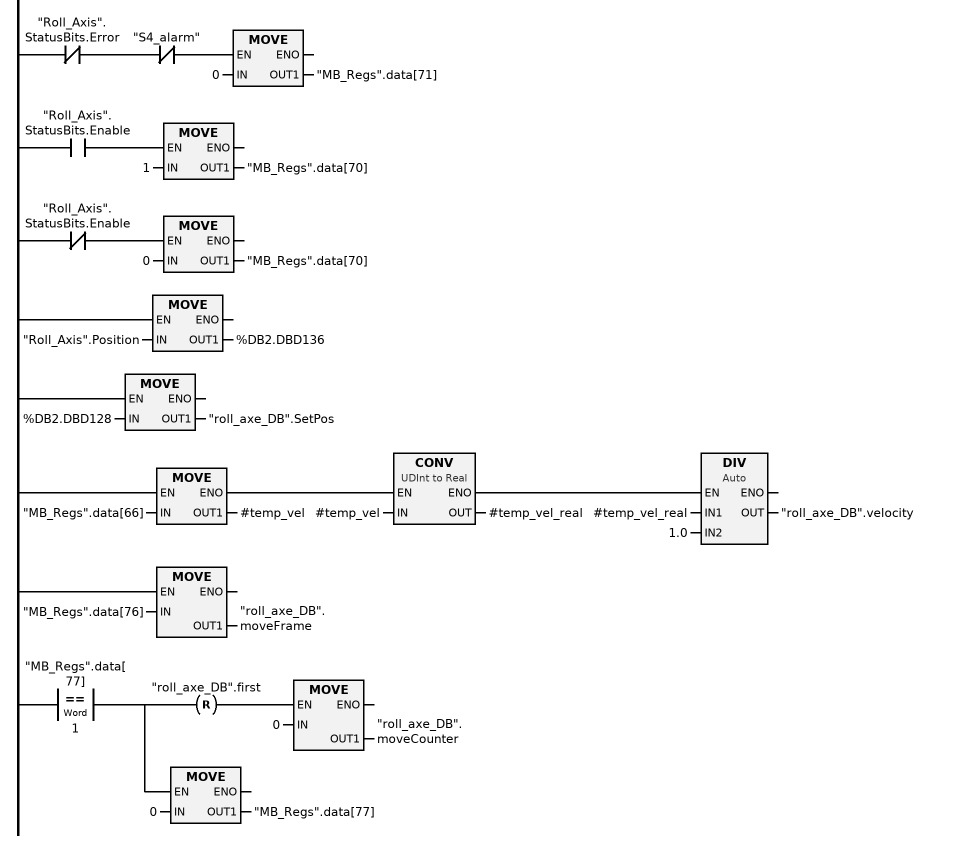
   RUNG wire#powerrail
      { S7_Templates := "SrcType := Word" } EQ_Contact(in1 := "MB_Regs".data[60], in2 := 1)
      Coil( "roll_axe_DB".axe1_motion_enable )
   END_RUNG
   RUNG wire#powerrail
      { S7_Templates := "SrcType := Word" } EQ_Contact(in1 := "MB_Regs".data[67], in2 := 1)
      wire#w1
      Coil( "roll_axe_DB".axe1_reset )
   END_RUNG
   RUNG wire#w1
      Move(in := 0, out1 => "MB_Regs".data[67])
   END_RUNG
   RUNG wire#powerrail
      { S7_Templates := "SrcType := Word" } EQ_Contact(in1 := "MB_Regs".data[61], in2 := 1)
      wire#w2
      Coil( "roll_axe_DB".axe1_home_execute )
   END_RUNG
   RUNG wire#w2
      Move(in := 0, out1 => "MB_Regs".data[61])
   END_RUNG
   RUNG wire#powerrail
      { S7_Templates := "SrcType := Word" } EQ_Contact(in1 := "MB_Regs".data[73], in2 := 1)
      wire#w3
      Coil( "roll_axe_DB".axe1_halt )
   END_RUNG
   RUNG wire#w3
      Move(in := 0, out1 => "MB_Regs".data[63])
   END_RUNG
   RUNG wire#powerrail
      { S7_Templates := "SrcType := Word" } EQ_Contact(in1 := "MB_Regs".data[75], in2 := 1)
      wire#w4
      Coil( "roll_axe_DB".axe1_move_relative_execute )
   END_RUNG
   RUNG wire#w4
      Move(in := 0, out1 => "MB_Regs".data[75])
   END_RUNG
   RUNG wire#powerrail
      { S7_Templates := "SrcType := Word" } EQ_Contact(in1 := "MB_Regs".data[62], in2 := 1)
      Coil( "roll_axe_DB".axe1_forward_execute )
   END_RUNG
   RUNG wire#powerrail
      { S7_Templates := "SrcType := Word" } EQ_Contact(in1 := "MB_Regs".data[63], in2 := 1)
      Coil( "roll_axe_DB".axe1_back_execute )
   END_RUNG
   RUNG wire#powerrail
      Contact( "Roll_Axis".StatusBits.HomingDone )
      Move(in := 1, out1 => "MB_Regs".data[72])
   END_RUNG
   RUNG wire#powerrail
      I_Contact( "Roll_Axis".StatusBits.HomingDone )
      Move(in := 0, out1 => "MB_Regs".data[72])
   END_RUNG
   RUNG wire#powerrail
      Contact( "Roll_Axis".StatusBits.Error )
      wire#w5
      Move(in := 1, out1 => "MB_Regs".data[71])
   END_RUNG
   RUNG wire#powerrail
      Contact( "S4_alarm" )
   END_RUNG wire#w5
   RUNG wire#powerrail
      I_Contact( "Roll_Axis".StatusBits.Error )
      I_Contact( "S4_alarm" )
      Move(in := 0, out1 => "MB_Regs".data[71])
   END_RUNG
   RUNG wire#powerrail
      Contact( "Roll_Axis".StatusBits.Enable )
      Move(in := 1, out1 => "MB_Regs".data[70])
   END_RUNG
   RUNG wire#powerrail
      I_Contact( "Roll_Axis".StatusBits.Enable )
      Move(in := 0, out1 => "MB_Regs".data[70])
   END_RUNG
   RUNG wire#powerrail
      Move(in := "Roll_Axis".Position, out1 => %DB2.DBD136)
   END_RUNG
   RUNG wire#powerrail
      Move(in := %DB2.DBD128, out1 => "roll_axe_DB".SetPos)
   END_RUNG
   RUNG wire#powerrail
      Move(in := "MB_Regs".data[66], out1 => #temp_vel)
      { S7_Templates := "[SrcType := UDInt, DestType := Real]" } Convert(in := #temp_vel, out => #temp_vel_real)
      Div(in1 := #temp_vel_real, in2 := 1.0, out => "roll_axe_DB".velocity)
   END_RUNG
   RUNG wire#powerrail
      Move(in := "MB_Regs".data[76], out1 => "roll_axe_DB".moveFrame)
   END_RUNG
   RUNG wire#powerrail
      { S7_Templates := "SrcType := Word" } EQ_Contact(in1 := "MB_Regs".data[77], in2 := 1)
      wire#w6
      R_Coil( "roll_axe_DB".first )
      Move(in := 0, out1 => "roll_axe_DB".moveCounter)
   END_RUNG
   RUNG wire#w6
      Move(in := 0, out1 => "MB_Regs".data[77])
   END_RUNG
   // the same network as SCL:
   "roll_axe_DB".axe1_motion_enable := "MB_Regs".data[60] = 1;
   "roll_axe_DB".axe1_reset := "MB_Regs".data[67] = 1;
   IF "roll_axe_DB".axe1_reset THEN "MB_Regs".data[67] := 0; END_IF;
   "roll_axe_DB".axe1_home_execute := "MB_Regs".data[61] = 1;
   IF "roll_axe_DB".axe1_home_execute THEN "MB_Regs".data[61] := 0; END_IF;
   "roll_axe_DB".axe1_halt := "MB_Regs".data[73] = 1;
   IF "roll_axe_DB".axe1_halt THEN "MB_Regs".data[63] := 0; END_IF;
   "roll_axe_DB".axe1_move_relative_execute := "MB_Regs".data[75] = 1;
   IF "roll_axe_DB".axe1_move_relative_execute THEN "MB_Regs".data[75] := 0; END_IF;
   "roll_axe_DB".axe1_forward_execute := "MB_Regs".data[62] = 1;
   "roll_axe_DB".axe1_back_execute := "MB_Regs".data[63] = 1;
   IF "Roll_Axis".StatusBits.HomingDone THEN "MB_Regs".data[72] := 1; END_IF;
   IF NOT "Roll_Axis".StatusBits.HomingDone THEN "MB_Regs".data[72] := 0; END_IF;
   IF "Roll_Axis".StatusBits.Error OR "S4_alarm" THEN "MB_Regs".data[71] := 1; END_IF;
   IF NOT "Roll_Axis".StatusBits.Error AND NOT "S4_alarm" THEN "MB_Regs".data[71] := 0; END_IF;
   IF "Roll_Axis".StatusBits.Enable THEN "MB_Regs".data[70] := 1; END_IF;
   IF NOT "Roll_Axis".StatusBits.Enable THEN "MB_Regs".data[70] := 0; END_IF;
   %DB2.DBD136 := "Roll_Axis".Position;
   "roll_axe_DB".SetPos := %DB2.DBD128;
   #temp_vel := "MB_Regs".data[66];
   #temp_vel_real := UDINT_TO_REAL(#temp_vel);
   "roll_axe_DB".velocity := #temp_vel_real / 1.0;
   "roll_axe_DB".moveFrame := "MB_Regs".data[76];
   IF "MB_Regs".data[77] = 1 THEN
       "roll_axe_DB".first := FALSE;
       "roll_axe_DB".moveCounter := 0;
       "MB_Regs".data[77] := 0;
   END_IF;
END_REGION
END_FUNCTION_BLOCK

FUNCTION_BLOCK "door_axe"   // FB2, LAD
{ S7_Optimized_Access := 'TRUE' }
VERSION : 0.1
   VAR
      SetPos : Real;
      velocity : Real;
      axe1_motion_enable : Bool;
      axe1_reset : Bool;
      axe1_halt : Bool;
      axe1_forward_execute : Bool;
      axe1_back_execute : Bool;
      axe1_home_execute : Bool;
      axe1_move_to_pos_execute : Bool;
      axe1_move_relative_execute : Bool;
      home_3_busy : Bool;
      home_0_busy : Bool;
      home_3_mode : Bool;
      home_0_mode : Bool;
      axe1_move_done : Bool;
      status : Bool;
   END_VAR
   VAR_TEMP
      temp_val2 : Real;
   END_VAR
   VAR CONSTANT
      vel_const : Real := 2.5;
   END_VAR
   VAR_TEMP   // added for the SCL form of the ladder/FBD networks
      _w1 : Bool;
   END_VAR
BEGIN

REGION Network 1
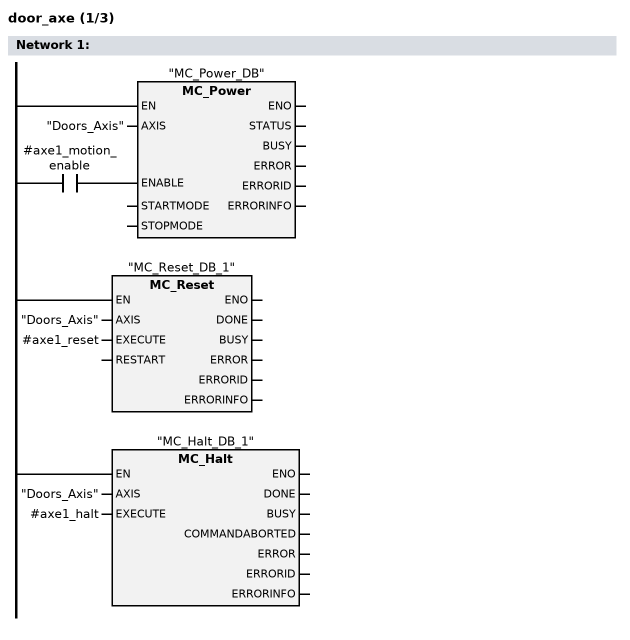
   "MC_Power_DB"(Axis := "Doors_Axis", Enable := #axe1_motion_enable);   // MC_Power
   "MC_Reset_DB_1"(Axis := "Doors_Axis", Execute := #axe1_reset);   // MC_Reset
   "MC_Halt_DB_1"(Axis := "Doors_Axis", Execute := #axe1_halt);   // MC_Halt
END_REGION

REGION Network 2
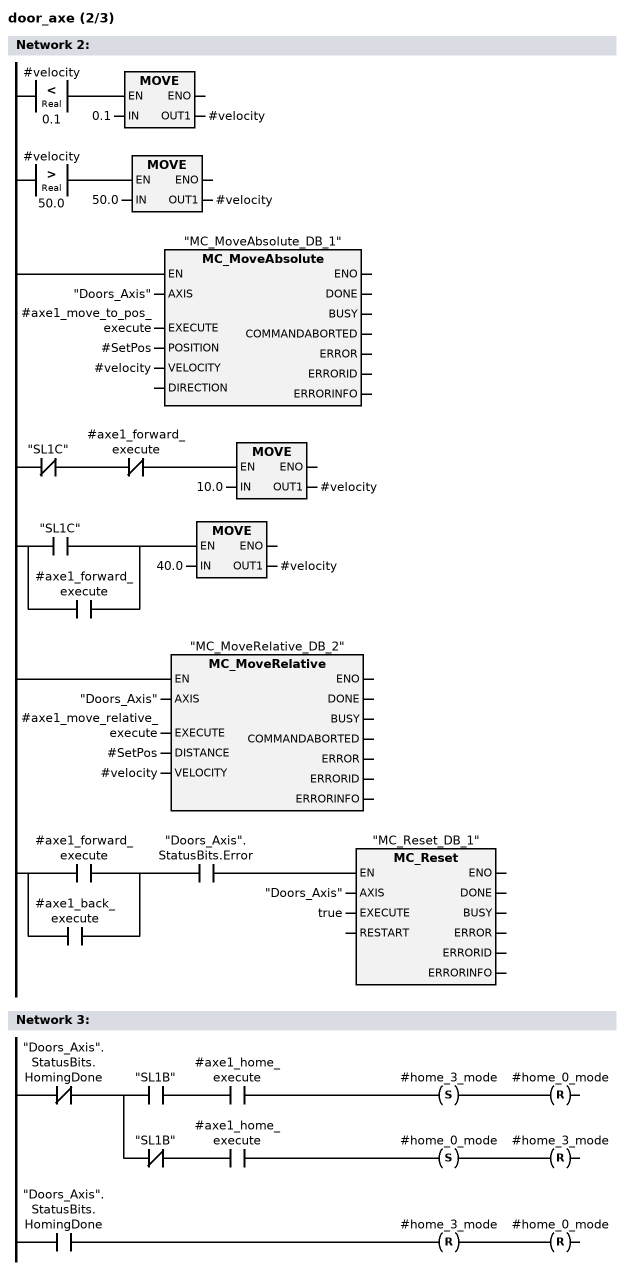
   IF #velocity < 0.1 THEN #velocity := 0.1; END_IF;
   IF #velocity > 50.0 THEN #velocity := 50.0; END_IF;
   "MC_MoveAbsolute_DB_1"(Axis := "Doors_Axis",   // MC_MoveAbsolute
                          Execute := #axe1_move_to_pos_execute,
                          Position := #SetPos,
                          Velocity := #velocity);
   IF NOT "SL1C" AND NOT #axe1_forward_execute THEN #velocity := 10.0; END_IF;
   IF "SL1C" OR #axe1_forward_execute THEN #velocity := 40.0; END_IF;
   "MC_MoveRelative_DB_2"(Axis := "Doors_Axis",   // MC_MoveRelative
                          Execute := #axe1_move_relative_execute,
                          Distance := #SetPos,
                          Velocity := #velocity);
   IF (#axe1_forward_execute OR #axe1_back_execute) AND "Doors_Axis".StatusBits.Error THEN
       "MC_Reset_DB_1"(Axis := "Doors_Axis", Execute := true);   // MC_Reset
   END_IF;
END_REGION

REGION Network 3
   RUNG wire#powerrail
      I_Contact( "Doors_Axis".StatusBits.HomingDone )
      wire#w1
      Contact( "SL1B" )
      Contact( #axe1_home_execute )
      S_Coil( #home_3_mode )
      R_Coil( #home_0_mode )
   END_RUNG
   RUNG wire#w1
      I_Contact( "SL1B" )
      Contact( #axe1_home_execute )
      S_Coil( #home_0_mode )
      R_Coil( #home_3_mode )
   END_RUNG
   RUNG wire#powerrail
      Contact( "Doors_Axis".StatusBits.HomingDone )
      R_Coil( #home_3_mode )
      R_Coil( #home_0_mode )
   END_RUNG
   // the same network as SCL:
   #_w1 := NOT "Doors_Axis".StatusBits.HomingDone;
   IF #_w1 AND "SL1B" AND #axe1_home_execute THEN
       #home_3_mode := TRUE;
       #home_0_mode := FALSE;
   END_IF;
   IF #_w1 AND NOT "SL1B" AND #axe1_home_execute THEN
       #home_0_mode := TRUE;
       #home_3_mode := FALSE;
   END_IF;
   IF "Doors_Axis".StatusBits.HomingDone THEN
       #home_3_mode := FALSE;
       #home_0_mode := FALSE;
   END_IF;
END_REGION

REGION Network 4: Ручная калибровка
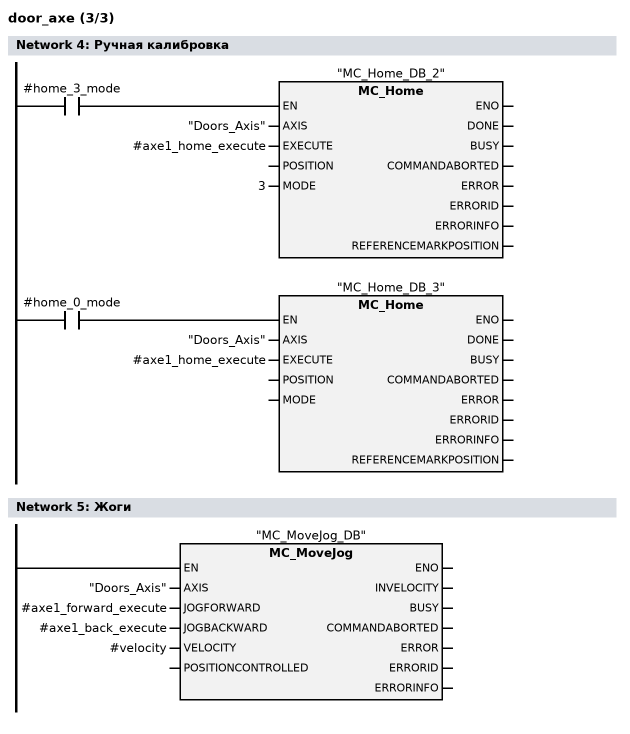
   IF #home_3_mode THEN
       "MC_Home_DB_2"(Axis := "Doors_Axis", Execute := #axe1_home_execute, Mode := 3);   // MC_Home
   END_IF;
   IF #home_0_mode THEN
       "MC_Home_DB_3"(Axis := "Doors_Axis", Execute := #axe1_home_execute);   // MC_Home
   END_IF;
END_REGION

REGION Network 5: Жоги
   "MC_MoveJog_DB"(Axis := "Doors_Axis",   // MC_MoveJog
                   JogForward := #axe1_forward_execute,
                   JogBackward := #axe1_back_execute,
                   Velocity := #velocity);
END_REGION
END_FUNCTION_BLOCK

FUNCTION_BLOCK "source_axe"   // FB3, LAD
{ S7_Optimized_Access := 'TRUE' }
VERSION : 0.1
   VAR
      SetPos : Real;
      velocity : Real;
      axe1_motion_enable : Bool;
      axe1_reset : Bool;
      axe1_halt : Bool;
      axe1_forward_execute : Bool;
      axe1_back_execute : Bool;
      axe1_home_execute : Bool;
      axe1_move_to_pos_execute : Bool;
      axe1_move_relative_execute : Bool;
      home_3_busy : Bool;
      home_0_busy : Bool;
      home_3_mode : Bool;
      home_0_mode : Bool;
      axe1_move_done : Bool;
      status : Bool;
   END_VAR
   VAR CONSTANT
      vel_const : Real := 2.5;
   END_VAR
   VAR_TEMP   // added for the SCL form of the ladder/FBD networks
      _w1 : Bool;
   END_VAR
BEGIN

REGION Network 1
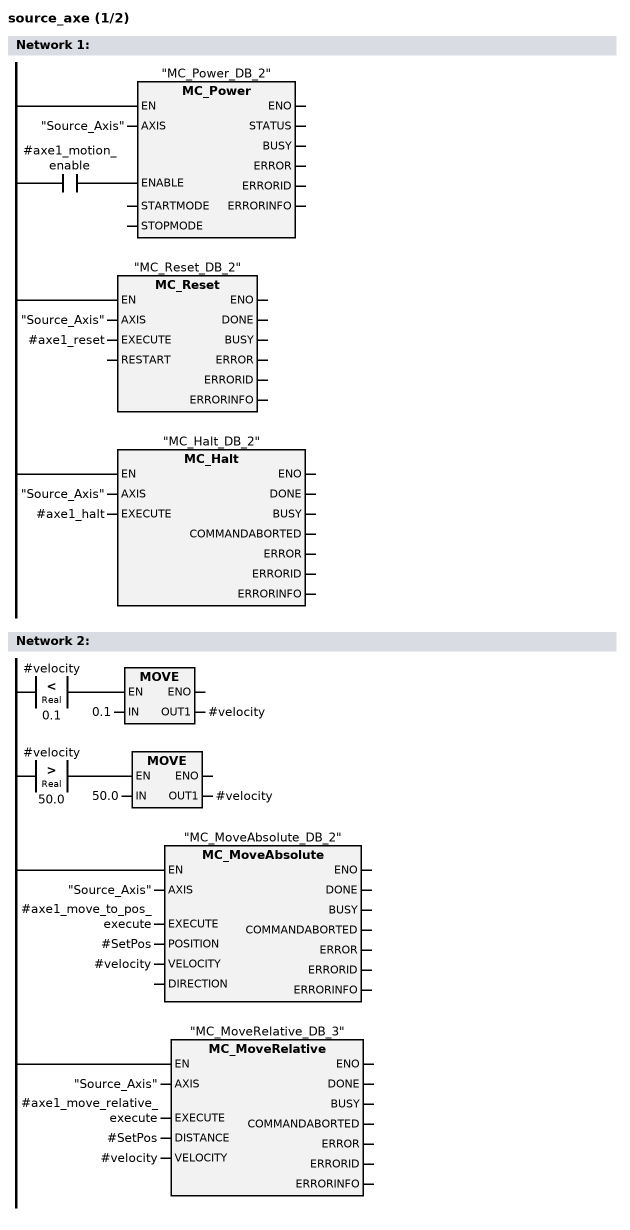
   "MC_Power_DB_2"(Axis := "Source_Axis", Enable := #axe1_motion_enable);   // MC_Power
   "MC_Reset_DB_2"(Axis := "Source_Axis", Execute := #axe1_reset);   // MC_Reset
   "MC_Halt_DB_2"(Axis := "Source_Axis", Execute := #axe1_halt);   // MC_Halt
END_REGION

REGION Network 2
   IF #velocity < 0.1 THEN #velocity := 0.1; END_IF;
   IF #velocity > 50.0 THEN #velocity := 50.0; END_IF;
   "MC_MoveAbsolute_DB_2"(Axis := "Source_Axis",   // MC_MoveAbsolute
                          Execute := #axe1_move_to_pos_execute,
                          Position := #SetPos,
                          Velocity := #velocity);
   "MC_MoveRelative_DB_3"(Axis := "Source_Axis",   // MC_MoveRelative
                          Execute := #axe1_move_relative_execute,
                          Distance := #SetPos,
                          Velocity := #velocity);
END_REGION

REGION Network 3
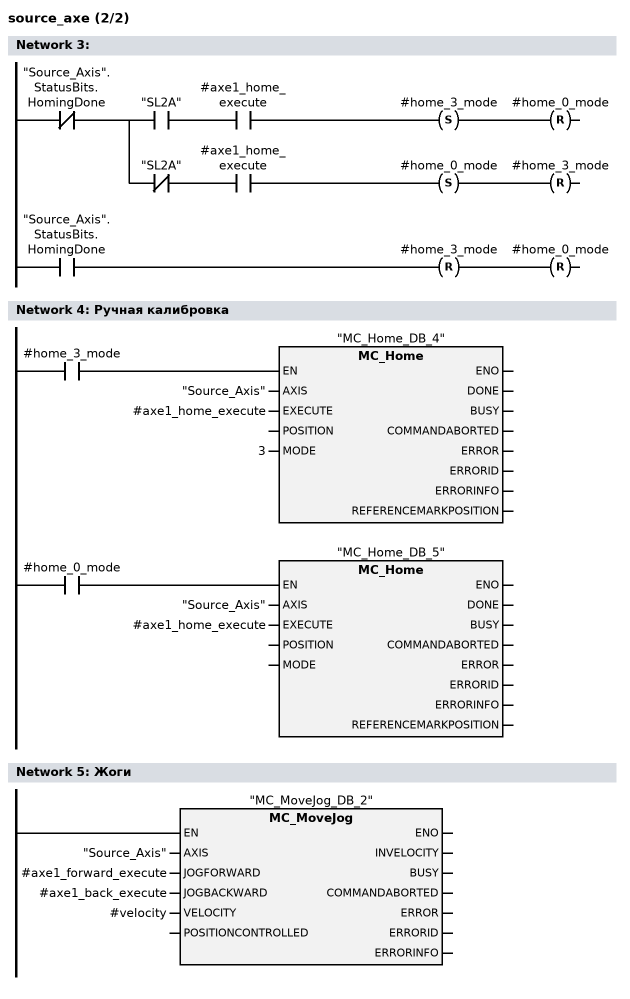
   RUNG wire#powerrail
      I_Contact( "Source_Axis".StatusBits.HomingDone )
      wire#w1
      Contact( "SL2A" )
      Contact( #axe1_home_execute )
      S_Coil( #home_3_mode )
      R_Coil( #home_0_mode )
   END_RUNG
   RUNG wire#w1
      I_Contact( "SL2A" )
      Contact( #axe1_home_execute )
      S_Coil( #home_0_mode )
      R_Coil( #home_3_mode )
   END_RUNG
   RUNG wire#powerrail
      Contact( "Source_Axis".StatusBits.HomingDone )
      R_Coil( #home_3_mode )
      R_Coil( #home_0_mode )
   END_RUNG
   // the same network as SCL:
   #_w1 := NOT "Source_Axis".StatusBits.HomingDone;
   IF #_w1 AND "SL2A" AND #axe1_home_execute THEN
       #home_3_mode := TRUE;
       #home_0_mode := FALSE;
   END_IF;
   IF #_w1 AND NOT "SL2A" AND #axe1_home_execute THEN
       #home_0_mode := TRUE;
       #home_3_mode := FALSE;
   END_IF;
   IF "Source_Axis".StatusBits.HomingDone THEN
       #home_3_mode := FALSE;
       #home_0_mode := FALSE;
   END_IF;
END_REGION

REGION Network 4: Ручная калибровка
   IF #home_3_mode THEN
       "MC_Home_DB_4"(Axis := "Source_Axis", Execute := #axe1_home_execute, Mode := 3);   // MC_Home
   END_IF;
   IF #home_0_mode THEN
       "MC_Home_DB_5"(Axis := "Source_Axis", Execute := #axe1_home_execute);   // MC_Home
   END_IF;
END_REGION

REGION Network 5: Жоги
   "MC_MoveJog_DB_2"(Axis := "Source_Axis",   // MC_MoveJog
                     JogForward := #axe1_forward_execute,
                     JogBackward := #axe1_back_execute,
                     Velocity := #velocity);
END_REGION
END_FUNCTION_BLOCK

FUNCTION_BLOCK "roll_axe"   // FB4, LAD
{ S7_Optimized_Access := 'TRUE' }
VERSION : 0.1
   VAR
      SetPos : Real;
      velocity : Real;
      axe1_motion_enable : Bool;
      axe1_reset : Bool;
      axe1_halt : Bool;
      axe1_forward_execute : Bool;
      axe1_back_execute : Bool;
      axe1_home_execute : Bool;
      axe1_move_to_pos_execute : Bool;
      axe1_move_relative_execute : Bool;
      home_3_busy : Bool;
      home_0_busy : Bool;
      home_3_mode : Bool;
      home_0_mode : Bool;
      axe1_move_done : Bool;
      status : Bool;
      moveCounter : Word;
      moveFrame : Word;
      moveCounter2 : Int;
      delayedEx : Bool;
      first : Bool;
   END_VAR
   VAR CONSTANT
      vel_const : Real := 2.5;
   END_VAR
   VAR_TEMP   // added for the SCL form of the ladder/FBD networks
      _w1 : Bool;
   END_VAR
BEGIN

REGION Network 1
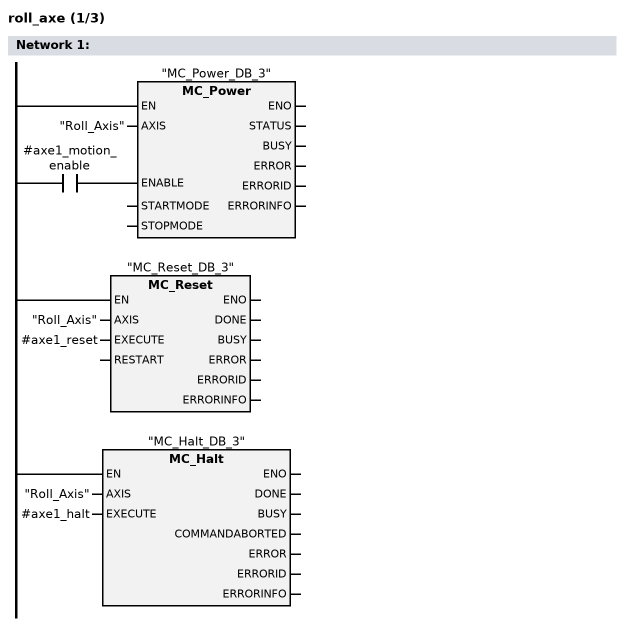
   "MC_Power_DB_3"(Axis := "Roll_Axis", Enable := #axe1_motion_enable);   // MC_Power
   "MC_Reset_DB_3"(Axis := "Roll_Axis", Execute := #axe1_reset);   // MC_Reset
   "MC_Halt_DB_3"(Axis := "Roll_Axis", Execute := #axe1_halt);   // MC_Halt
END_REGION

REGION Network 2
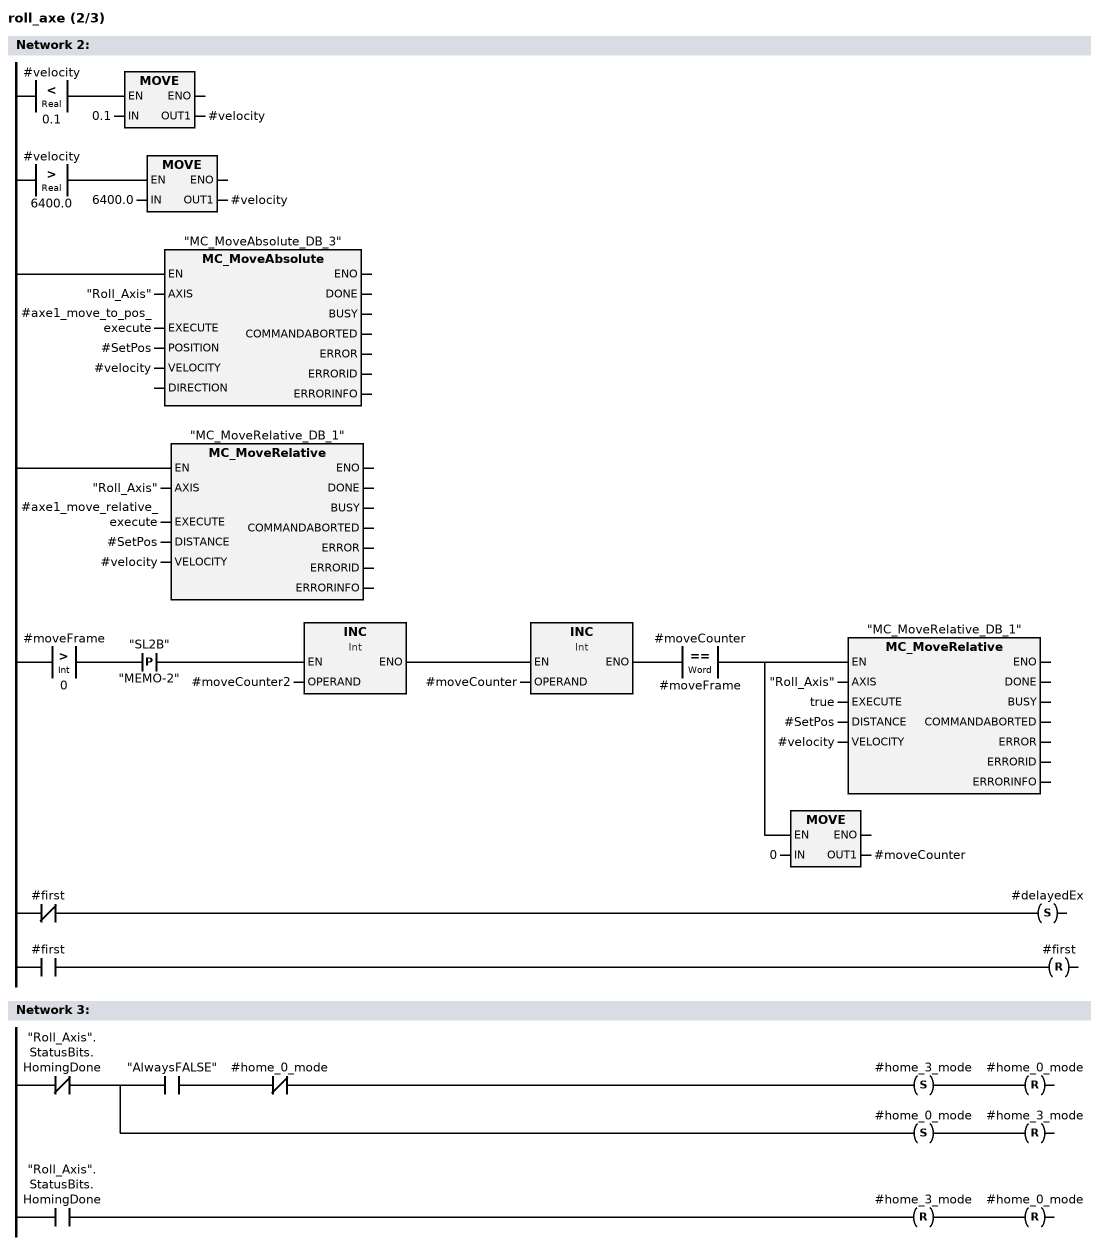
   IF #velocity < 0.1 THEN #velocity := 0.1; END_IF;
   IF #velocity > 6400.0 THEN #velocity := 6400.0; END_IF;
   "MC_MoveAbsolute_DB_3"(Axis := "Roll_Axis",   // MC_MoveAbsolute
                          Execute := #axe1_move_to_pos_execute,
                          Position := #SetPos,
                          Velocity := #velocity);
   "MC_MoveRelative_DB_1"(Axis := "Roll_Axis",   // MC_MoveRelative
                          Execute := #axe1_move_relative_execute,
                          Distance := #SetPos,
                          Velocity := #velocity);
   #_w1 := (#moveFrame > 0) AND "SL2B" AND NOT "MEMO-2";   // rising edge of "SL2B"
   "MEMO-2" := "SL2B";
   IF #_w1 THEN
       #moveCounter2 := #moveCounter2 + 1;
       #moveCounter := #moveCounter + 1;
   END_IF;
   IF #_w1 AND (#moveCounter = #moveFrame) THEN
       "MC_MoveRelative_DB_1"(Axis := "Roll_Axis", Execute := true, Distance := #SetPos, Velocity := #velocity);   // MC_MoveRelative
       #moveCounter := 0;
   END_IF;
   IF NOT #first THEN #delayedEx := TRUE; END_IF;
   IF #first THEN #first := FALSE; END_IF;
END_REGION

REGION Network 3
   RUNG wire#powerrail
      I_Contact( "Roll_Axis".StatusBits.HomingDone )
      wire#w1
      Contact( "AlwaysFALSE" )
      I_Contact( #home_0_mode )
      S_Coil( #home_3_mode )
      R_Coil( #home_0_mode )
   END_RUNG
   RUNG wire#w1
      S_Coil( #home_0_mode )
      R_Coil( #home_3_mode )
   END_RUNG
   RUNG wire#powerrail
      Contact( "Roll_Axis".StatusBits.HomingDone )
      R_Coil( #home_3_mode )
      R_Coil( #home_0_mode )
   END_RUNG
   // the same network as SCL:
   #_w1 := NOT "Roll_Axis".StatusBits.HomingDone;
   IF #_w1 AND "AlwaysFALSE" AND NOT #home_0_mode THEN
       #home_3_mode := TRUE;
       #home_0_mode := FALSE;
   END_IF;
   IF #_w1 THEN
       #home_0_mode := TRUE;
       #home_3_mode := FALSE;
   END_IF;
   IF "Roll_Axis".StatusBits.HomingDone THEN
       #home_3_mode := FALSE;
       #home_0_mode := FALSE;
   END_IF;
END_REGION

REGION Network 4: Ручная калибровка
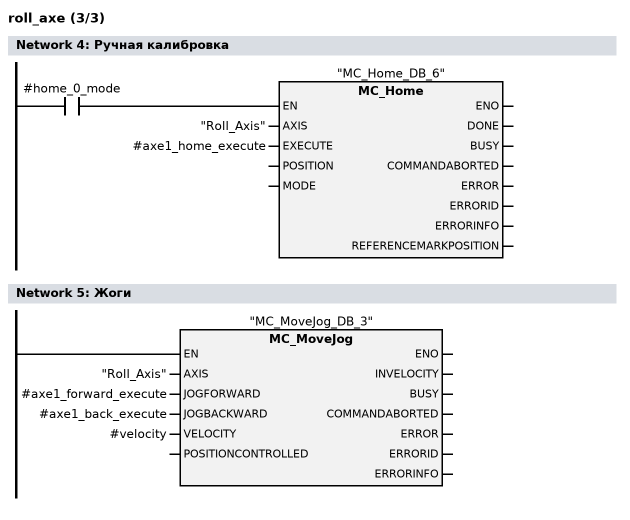
   IF #home_0_mode THEN
       "MC_Home_DB_6"(Axis := "Roll_Axis", Execute := #axe1_home_execute);   // MC_Home
   END_IF;
END_REGION

REGION Network 5: Жоги
   "MC_MoveJog_DB_3"(Axis := "Roll_Axis",   // MC_MoveJog
                     JogForward := #axe1_forward_execute,
                     JogBackward := #axe1_back_execute,
                     Velocity := #velocity);
END_REGION
END_FUNCTION_BLOCK

FUNCTION_BLOCK "safety"   // FB5, LAD
{ S7_Optimized_Access := 'TRUE' }
VERSION : 0.1
BEGIN

REGION Network 1: блокировка излучекеия при открытом периметри
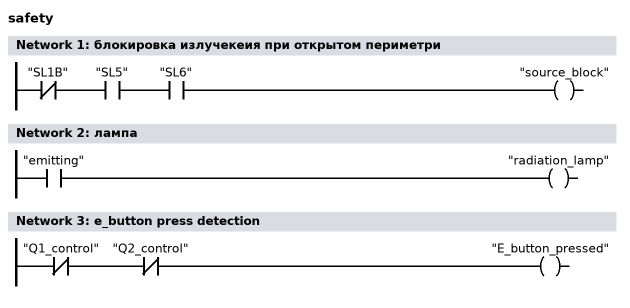
   RUNG wire#powerrail
      I_Contact( "SL1B" )
      Contact( "SL5" )
      Contact( "SL6" )
      Coil( "source_block" )
   END_RUNG
   // the same network as SCL:
   "source_block" := NOT "SL1B" AND "SL5" AND "SL6";
END_REGION

REGION Network 2: лампа
   RUNG wire#powerrail
      Contact( "emitting" )
      Coil( "radiation_lamp" )
   END_RUNG
   // the same network as SCL:
   "radiation_lamp" := "emitting";
END_REGION

REGION Network 3: e_button press detection
   RUNG wire#powerrail
      I_Contact( "Q1_control" )
      I_Contact( "Q2_control" )
      Coil( "E_button_pressed" )
   END_RUNG
   // the same network as SCL:
   "E_button_pressed" := NOT "Q1_control" AND NOT "Q2_control";
END_REGION
END_FUNCTION_BLOCK

FUNCTION_BLOCK "detector_axe"   // FB12, LAD
{ S7_Optimized_Access := 'TRUE' }
VERSION : 0.1
   VAR
      SetPos : Real;
      velocity : Real;
      axe1_motion_enable : Bool;
      axe1_reset : Bool;
      axe1_halt : Bool;
      axe1_forward_execute : Bool;
      axe1_back_execute : Bool;
      axe1_home_execute : Bool;
      axe1_move_to_pos_execute : Bool;
      axe1_move_relative_execute : Bool;
      home_3_busy : Bool;
      home_0_busy : Bool;
      home_3_mode : Bool;
      home_0_mode : Bool;
      axe1_move_done : Bool;
      status : Bool;
   END_VAR
   VAR CONSTANT
      vel_const : Real := 2.5;
   END_VAR
   VAR_TEMP   // added for the SCL form of the ladder/FBD networks
      _w1 : Bool;
   END_VAR
BEGIN

REGION Network 1
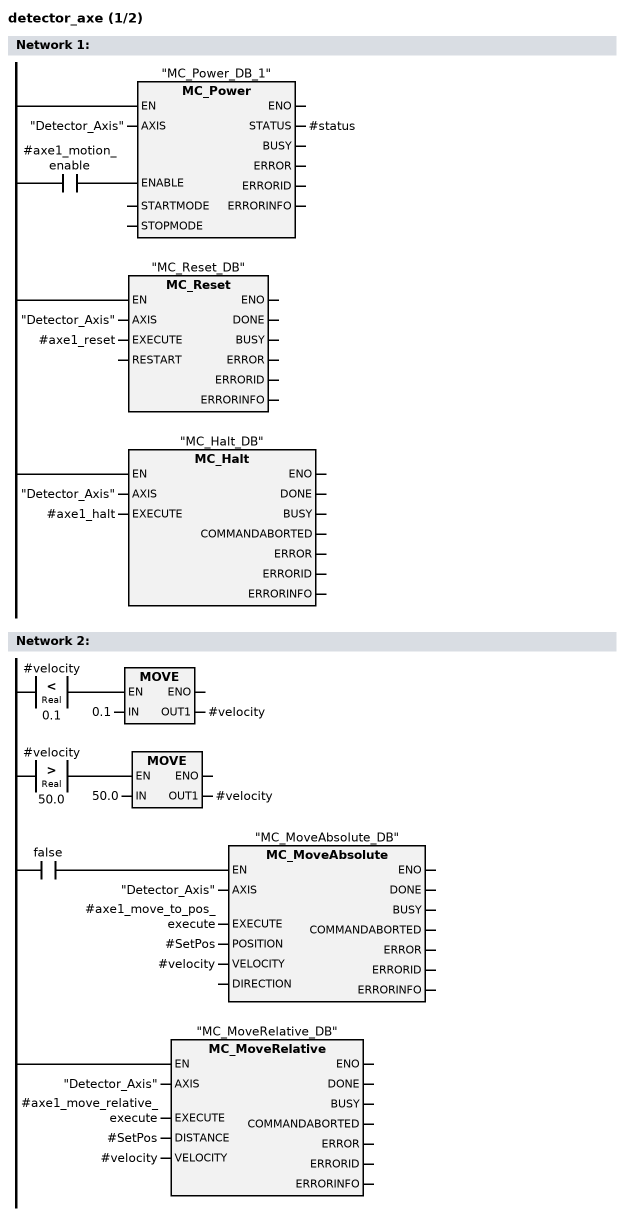
   "MC_Power_DB_1"(Axis := "Detector_Axis", Enable := #axe1_motion_enable, Status => #status);   // MC_Power
   "MC_Reset_DB"(Axis := "Detector_Axis", Execute := #axe1_reset);   // MC_Reset
   "MC_Halt_DB"(Axis := "Detector_Axis", Execute := #axe1_halt);   // MC_Halt
END_REGION

REGION Network 2
   IF #velocity < 0.1 THEN #velocity := 0.1; END_IF;
   IF #velocity > 50.0 THEN #velocity := 50.0; END_IF;
   IF false THEN
       "MC_MoveAbsolute_DB"(Axis := "Detector_Axis",   // MC_MoveAbsolute
                            Execute := #axe1_move_to_pos_execute,
                            Position := #SetPos,
                            Velocity := #velocity);
   END_IF;
   "MC_MoveRelative_DB"(Axis := "Detector_Axis",   // MC_MoveRelative
                        Execute := #axe1_move_relative_execute,
                        Distance := #SetPos,
                        Velocity := #velocity);
END_REGION

REGION Network 3
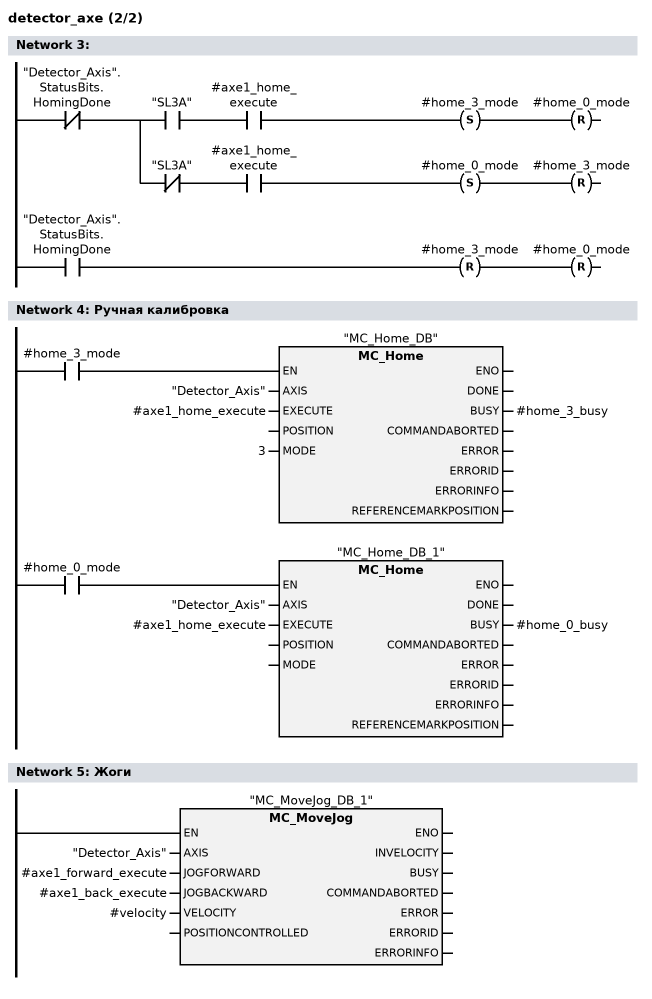
   RUNG wire#powerrail
      I_Contact( "Detector_Axis".StatusBits.HomingDone )
      wire#w1
      Contact( "SL3A" )
      Contact( #axe1_home_execute )
      S_Coil( #home_3_mode )
      R_Coil( #home_0_mode )
   END_RUNG
   RUNG wire#w1
      I_Contact( "SL3A" )
      Contact( #axe1_home_execute )
      S_Coil( #home_0_mode )
      R_Coil( #home_3_mode )
   END_RUNG
   RUNG wire#powerrail
      Contact( "Detector_Axis".StatusBits.HomingDone )
      R_Coil( #home_3_mode )
      R_Coil( #home_0_mode )
   END_RUNG
   // the same network as SCL:
   #_w1 := NOT "Detector_Axis".StatusBits.HomingDone;
   IF #_w1 AND "SL3A" AND #axe1_home_execute THEN
       #home_3_mode := TRUE;
       #home_0_mode := FALSE;
   END_IF;
   IF #_w1 AND NOT "SL3A" AND #axe1_home_execute THEN
       #home_0_mode := TRUE;
       #home_3_mode := FALSE;
   END_IF;
   IF "Detector_Axis".StatusBits.HomingDone THEN
       #home_3_mode := FALSE;
       #home_0_mode := FALSE;
   END_IF;
END_REGION

REGION Network 4: Ручная калибровка
   IF #home_3_mode THEN
       "MC_Home_DB"(Axis := "Detector_Axis", Execute := #axe1_home_execute, Mode := 3, Busy => #home_3_busy);   // MC_Home
   END_IF;
   IF #home_0_mode THEN
       "MC_Home_DB_1"(Axis := "Detector_Axis", Execute := #axe1_home_execute, Busy => #home_0_busy);   // MC_Home
   END_IF;
END_REGION

REGION Network 5: Жоги
   "MC_MoveJog_DB_1"(Axis := "Detector_Axis",   // MC_MoveJog
                     JogForward := #axe1_forward_execute,
                     JogBackward := #axe1_back_execute,
                     Velocity := #velocity);
END_REGION
END_FUNCTION_BLOCK

FUNCTION "ProcessCalibrationStatus" : Void   // FC1, LAD
{ S7_Optimized_Access := 'TRUE' }
VERSION : 0.1
BEGIN

REGION Network 1
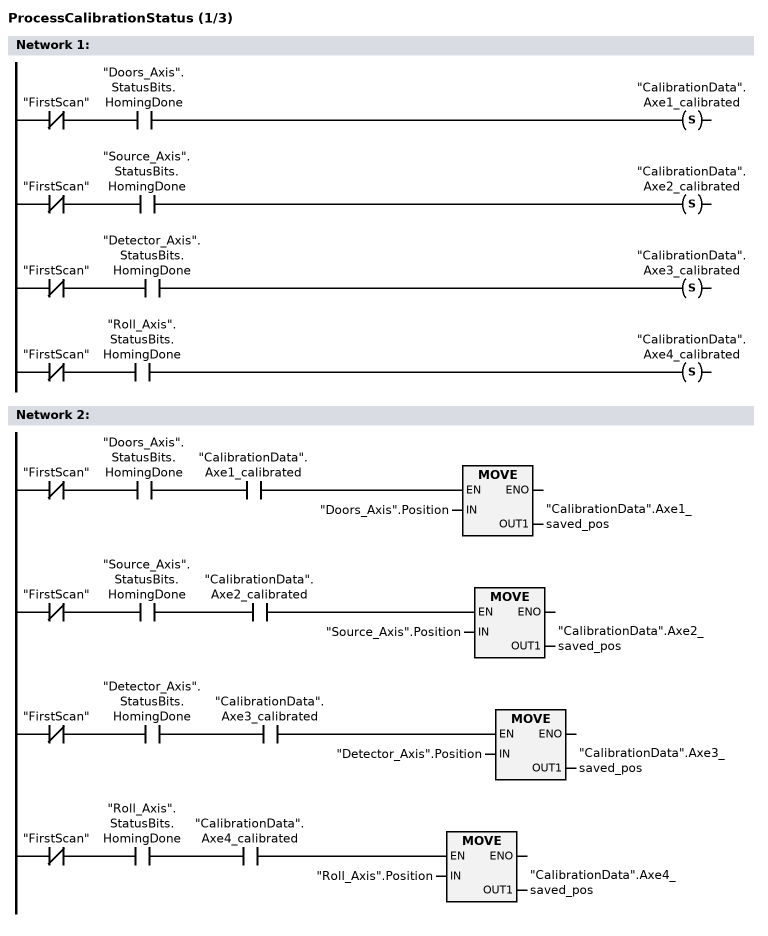
   RUNG wire#powerrail
      I_Contact( "FirstScan" )
      Contact( "Doors_Axis".StatusBits.HomingDone )
      S_Coil( "CalibrationData".Axe1_calibrated )
   END_RUNG
   RUNG wire#powerrail
      I_Contact( "FirstScan" )
      Contact( "Source_Axis".StatusBits.HomingDone )
      S_Coil( "CalibrationData".Axe2_calibrated )
   END_RUNG
   RUNG wire#powerrail
      I_Contact( "FirstScan" )
      Contact( "Detector_Axis".StatusBits.HomingDone )
      S_Coil( "CalibrationData".Axe3_calibrated )
   END_RUNG
   RUNG wire#powerrail
      I_Contact( "FirstScan" )
      Contact( "Roll_Axis".StatusBits.HomingDone )
      S_Coil( "CalibrationData".Axe4_calibrated )
   END_RUNG
   // the same network as SCL:
   IF NOT "FirstScan" AND "Doors_Axis".StatusBits.HomingDone THEN
       "CalibrationData".Axe1_calibrated := TRUE;
   END_IF;
   IF NOT "FirstScan" AND "Source_Axis".StatusBits.HomingDone THEN
       "CalibrationData".Axe2_calibrated := TRUE;
   END_IF;
   IF NOT "FirstScan" AND "Detector_Axis".StatusBits.HomingDone THEN
       "CalibrationData".Axe3_calibrated := TRUE;
   END_IF;
   IF NOT "FirstScan" AND "Roll_Axis".StatusBits.HomingDone THEN
       "CalibrationData".Axe4_calibrated := TRUE;
   END_IF;
END_REGION

REGION Network 2
   RUNG wire#powerrail
      I_Contact( "FirstScan" )
      Contact( "Doors_Axis".StatusBits.HomingDone )
      Contact( "CalibrationData".Axe1_calibrated )
      Move(in := "Doors_Axis".Position, out1 => "CalibrationData".Axe1_saved_pos)
   END_RUNG
   RUNG wire#powerrail
      I_Contact( "FirstScan" )
      Contact( "Source_Axis".StatusBits.HomingDone )
      Contact( "CalibrationData".Axe2_calibrated )
      Move(in := "Source_Axis".Position, out1 => "CalibrationData".Axe2_saved_pos)
   END_RUNG
   RUNG wire#powerrail
      I_Contact( "FirstScan" )
      Contact( "Detector_Axis".StatusBits.HomingDone )
      Contact( "CalibrationData".Axe3_calibrated )
      Move(in := "Detector_Axis".Position, out1 => "CalibrationData".Axe3_saved_pos)
   END_RUNG
   RUNG wire#powerrail
      I_Contact( "FirstScan" )
      Contact( "Roll_Axis".StatusBits.HomingDone )
      Contact( "CalibrationData".Axe4_calibrated )
      Move(in := "Roll_Axis".Position, out1 => "CalibrationData".Axe4_saved_pos)
   END_RUNG
   // the same network as SCL:
   IF NOT "FirstScan" AND "Doors_Axis".StatusBits.HomingDone AND "CalibrationData".Axe1_calibrated THEN
       "CalibrationData".Axe1_saved_pos := "Doors_Axis".Position;
   END_IF;
   IF NOT "FirstScan" AND "Source_Axis".StatusBits.HomingDone AND "CalibrationData".Axe2_calibrated THEN
       "CalibrationData".Axe2_saved_pos := "Source_Axis".Position;
   END_IF;
   IF NOT "FirstScan" AND "Detector_Axis".StatusBits.HomingDone AND "CalibrationData".Axe3_calibrated THEN
       "CalibrationData".Axe3_saved_pos := "Detector_Axis".Position;
   END_IF;
   IF NOT "FirstScan" AND "Roll_Axis".StatusBits.HomingDone AND "CalibrationData".Axe4_calibrated THEN
       "CalibrationData".Axe4_saved_pos := "Roll_Axis".Position;
   END_IF;
END_REGION

REGION Network 3
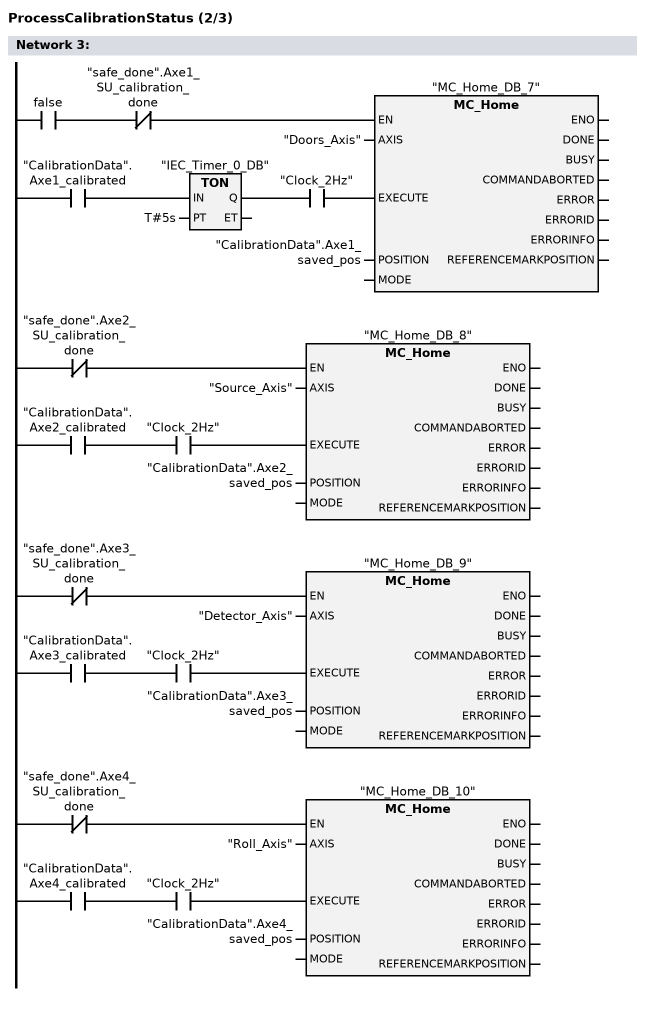
   "IEC_Timer_0_DB".TON(IN := "CalibrationData".Axe1_calibrated, PT := T#5s);
   IF false AND NOT "safe_done".Axe1_SU_calibration_done THEN
       "MC_Home_DB_7"(Axis := "Doors_Axis",   // MC_Home
                      Execute := "IEC_Timer_0_DB".Q AND "Clock_2Hz",
                      Position := "CalibrationData".Axe1_saved_pos);
   END_IF;
   IF NOT "safe_done".Axe2_SU_calibration_done THEN
       "MC_Home_DB_8"(Axis := "Source_Axis",   // MC_Home
                      Execute := "CalibrationData".Axe2_calibrated AND "Clock_2Hz",
                      Position := "CalibrationData".Axe2_saved_pos);
   END_IF;
   IF NOT "safe_done".Axe3_SU_calibration_done THEN
       "MC_Home_DB_9"(Axis := "Detector_Axis",   // MC_Home
                      Execute := "CalibrationData".Axe3_calibrated AND "Clock_2Hz",
                      Position := "CalibrationData".Axe3_saved_pos);
   END_IF;
   IF NOT "safe_done".Axe4_SU_calibration_done THEN
       "MC_Home_DB_10"(Axis := "Roll_Axis",   // MC_Home
                       Execute := "CalibrationData".Axe4_calibrated AND "Clock_2Hz",
                       Position := "CalibrationData".Axe4_saved_pos);
   END_IF;
END_REGION

REGION Network 4
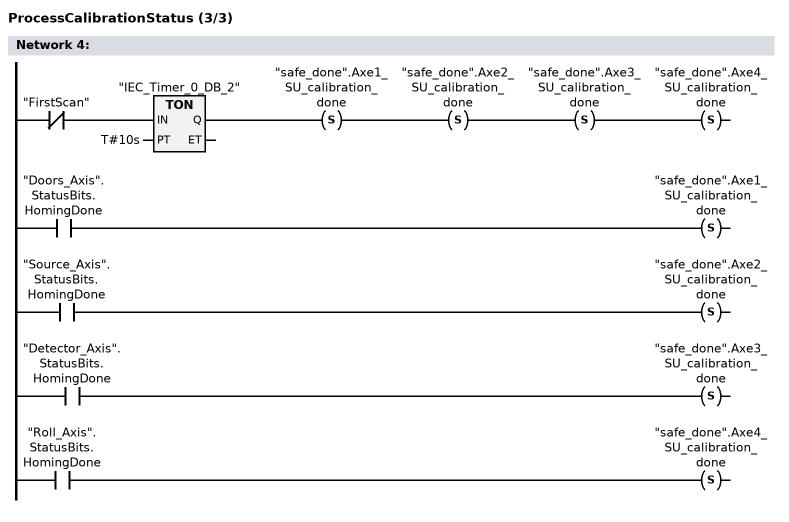
   "IEC_Timer_0_DB_2".TON(IN := NOT "FirstScan", PT := T#10s);
   IF "IEC_Timer_0_DB_2".Q THEN
       "safe_done".Axe1_SU_calibration_done := TRUE;
       "safe_done".Axe2_SU_calibration_done := TRUE;
       "safe_done".Axe3_SU_calibration_done := TRUE;
       "safe_done".Axe4_SU_calibration_done := TRUE;
   END_IF;
   IF "Doors_Axis".StatusBits.HomingDone THEN "safe_done".Axe1_SU_calibration_done := TRUE; END_IF;
   IF "Source_Axis".StatusBits.HomingDone THEN "safe_done".Axe2_SU_calibration_done := TRUE; END_IF;
   IF "Detector_Axis".StatusBits.HomingDone THEN "safe_done".Axe3_SU_calibration_done := TRUE; END_IF;
   IF "Roll_Axis".StatusBits.HomingDone THEN "safe_done".Axe4_SU_calibration_done := TRUE; END_IF;
END_REGION
END_FUNCTION

ORGANIZATION_BLOCK "Main"   // OB1, LAD, ProgramCycle
TITLE = "Main Program Sweep (Cycle)"
{ S7_Optimized_Access := 'TRUE' }
VERSION : 0.1
   VAR_INPUT
      Initial_Call : Bool;   // Initial call of this OB
      Remanence : Bool;   // =True, if remanent data are available
   END_VAR
BEGIN

REGION Network 1
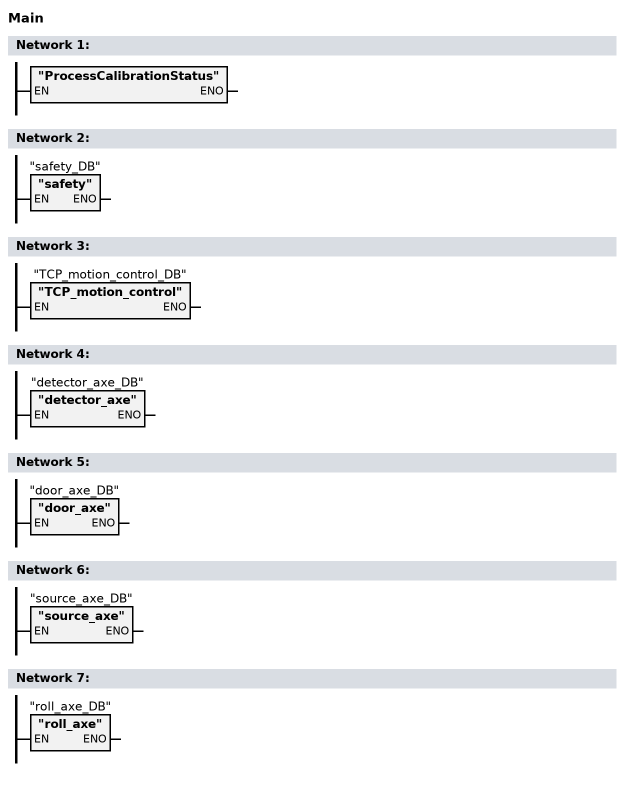
   RUNG wire#powerrail
      "ProcessCalibrationStatus"()
   END_RUNG
   // the same network as SCL:
   "ProcessCalibrationStatus"();
END_REGION

REGION Network 2
   RUNG wire#powerrail
      "safety_DB"()
   END_RUNG
   // the same network as SCL:
   "safety_DB"();   // "safety"
END_REGION

REGION Network 3
   RUNG wire#powerrail
      "TCP_motion_control_DB"()
   END_RUNG
   // the same network as SCL:
   "TCP_motion_control_DB"();   // "TCP_motion_control"
END_REGION

REGION Network 4
   RUNG wire#powerrail
      "detector_axe_DB"()
   END_RUNG
   // the same network as SCL:
   "detector_axe_DB"();   // "detector_axe"
END_REGION

REGION Network 5
   RUNG wire#powerrail
      "door_axe_DB"()
   END_RUNG
   // the same network as SCL:
   "door_axe_DB"();   // "door_axe"
END_REGION

REGION Network 6
   RUNG wire#powerrail
      "source_axe_DB"()
   END_RUNG
   // the same network as SCL:
   "source_axe_DB"();   // "source_axe"
END_REGION

REGION Network 7
   RUNG wire#powerrail
      "roll_axe_DB"()
   END_RUNG
   // the same network as SCL:
   "roll_axe_DB"();   // "roll_axe"
END_REGION
END_ORGANIZATION_BLOCK